	3410:
		stFolderCom.TaskBackGauge	:=eTask_BackGauge_AbsPos;
		stFolderCom.paraBackGauge	:=stFolder.BackGauge_M_ActPos+10;
		iSemiAutoStp	:=3411;
	3411:
		SA_Ton2(IN:=stFolderCom.TaskBackGauge = eTask_NULL , PT:=T#100MS , Q=> , ET=> );
		IF SA_Ton2.Q THEN
			SA_Ton2(IN:=FALSE);
			iSemiAutoStp	:=3420;
		END_IF	
	3420:
		stFolderCom.TaskClamp	:=eTask_ClampUnlock;
		stFolderCom.paraClamp	:=1;
		iSemiAutoStp	:=3421;
	3421:
		IF stFolderCom.TaskClamp = eTask_NULL THEN
			iSemiAutoStp	:=350;
		END_IF
		*)
(********************************************************************************)
	350:
		stFolderCom.TaskBackGauge	:=eTask_BackGauge_AbsPos;
		_ActBG_Target				:=SemiAuto_ActJob.BackGaugePos;
		stFolderCom.paraBackGaugeVelo	:= CNST_BACKGAUGE_SPEED_LOW;
		iSemiAutoStp	:=351;
	351:
		IF stFolderCom.TaskBackGauge = eTask_NULL THEN
			iSemiAutoStp	:=360;
		END_IF
	360:
		stFolderCom.TaskApron	:=eTask_ApronBtmFold_AbsPos;
		stFolderCom.ParaApronBtmFold	:=180;
		stFolderCom.paraApronFold_Auto	:=FALSE;
		iSemiAutoStp	:=361;
	361:
		IF stFolderCom.TaskApron = eTask_NULL THEN
			iSemiAutoStp	:=362;
		END_IF
	362:
		IF stFolder.Status.ApronBtmFold_AtHome THEN
			iSemiAutoStp	:=363;
		END_IF;
	363:
		stFolderCom.TaskClamp	:=eTask_ClampJog;
		IF _Contius OR (NOT _Contius AND rtPdlFold.Q) THEN
			iSemiAutoStp	:=370;
		END_IF
	370:
		//Out_GripperDatum_S0	:=Out_GripperDatum_S1	:=TRUE;		//insert to UNIT
		stFolderCom.TaskClamp	:=eTask_ClampLock;
		stFolderCom.paraClamp	:=6;
		iSemiAutoStp	:=371;
	371:
		IF stFolderCom.TaskClamp = eTask_NULL THEN
			iSemiAutoStp	:=372;
		END_IF
	372:
		IF SemiAuto_ActJob.ActType=1 THEN		//Close Squash
			iSemiAutoStp	:=380;
		ELSIF SemiAuto_ActJob.ActType=2 THEN	//Open Squash
			iSemiAutoStp	:=3800;
		END_IF
	380:
		ton372(IN:=TRUE , PT:=T#300MS , Q=> , ET=> );
		IF ton372.Q THEN
			iSemiAutoStp	:=500;
			ton372(IN:=FALSE);
		END_IF;
	//Open Squash Fun. 3800-3830
	3800:
		stFolderCom.TaskClamp	:=eTask_ClampUnlock;
		stFolderCom.paraClamp	:=1;
		iSemiAutoStp	:=3801;
	3801:
		IF stFolderCom.TaskClamp = eTask_NULL AND stFolder.ClampHt_ActPos>=stFolderPara.Clamp_MidPos  THEN
			iSemiAutoStp	:=3810;
		END_IF
	3810:
		stFolderCom.TaskBackGauge	:=eTask_BackGauge_AbsPos;
		IF SemiAuto_ActJob.FoldDir=0 THEN
			_tmp0	:=stFolderPara.SquashBackstop_OpenTop;
		ELSE
			_tmp0	:=stFolderPara.SquashBackstop_OpenBtm;
		END_IF
		_ActBG_Target				:=SemiAuto_ActJob.BackGaugePos-stFolderPara.SquashBackstop_External-_tmp0;
		stFolderCom.paraBackGaugeVelo	:= CNST_BACKGAUGE_SPEED_LOW;
		iSemiAutoStp	:=3811;
	3811:
		IF stFolderCom.TaskBackGauge = eTask_NULL THEN
			iSemiAutoStp	:=3820;
		END_IF
	3820:
		stFolderCom.TaskClamp	:=eTask_ClampLock;
		stFolderCom.paraClamp	:=6;
		iSemiAutoStp	:=3821;
	3821:
		IF stFolderCom.TaskClamp = eTask_NULL THEN
			iSemiAutoStp	:=380;
		END_IF


(*--------------------------------------------------------------------------*)
(*------------------------------分条功能开始--------------------------------*)	
(*--------------------------------------------------------------------------*)
	400:
	IF Hmi_bArray[62] THEN			//分条  + Slitter S.W.
		iSemiAutoStp	:=401;
	ELSE
		iSemiAutoStp	:=500;
	END_IF
	401:
		stFolderCom.TaskClamp	:=eTask_ClampJog;
		stFolder.SlitterRef		:=TRUE;
		IF stFolder.ClampHt_ActPos > stFolderPara.ClampHalfPos THEN
			stFolderCom.TaskBackGauge	:=eTask_BackGauge_AbsPos;
			_ActBG_Target				:=SemiAuto_ActJob.BackGaugePos;
			stFolderCom.paraBackGauge_GripType	:=SemiAuto_ActJob.GripType;
			stFolderCom.paraBackGaugeVelo	:= CNST_BACKGAUGE_SPEED_HIGH;
			bGripperDatumBack:=TRUE;
			iSemiAutoStp	:=402;
		END_IF
	402:
		IF stFolderCom.TaskBackGauge=eTask_NULL THEN
			iSemiAutoStp	:=410;
		END_IF
	410:
		Hmi_iArray[22]:=2 ;				//msg： Lock Grip
		IF stFolder.Status.Gripper THEN
			Hmi_iArray[22]:=0 ;
			iSemiAutoStp	:=420;
		END_IF;
	420:
		//Out_GripperDatum_S0	:=Out_GripperDatum_S1	:=TRUE;		//insert to UNIT
		stFolderCom.TaskClamp	:=eTask_ClampLock;
		stFolderCom.paraClamp	:=6;
		IF stFolder.Status.Clamp_AtPressPoint THEN
			iSemiAutoStp	:=430;
		END_IF
	430:
		stFolderCom.ParaApronBtmSlide := 0;
		stFolderCom.ParaApronTopSlide := 3;
		stFolderCom.TaskApron	:=eTask_ApronDaulSlide_AbsPos;
		iSemiAutoStp	:=431;
	431:
		IF stFolderCom.TaskApron = eTask_NULL THEN
			iSemiAutoStp	:=440;
		END_IF
	440:
		Hmi_iArray[22]:=7;				//msg： Operator Slitter
		stFolderCom.TaskSlitter	:=eTask_SlitterAct;
		iSemiAutoStp	:=441;
	441:
		IF stFolderCom.TaskSlitter	= eTask_NULL THEN
			iSemiAutoStp	:=450;
			Hmi_iArray[22]:=0;	
		END_IF
	450:
		stFolder.SlitterRef		:=FALSE;
		iSemiAutoStp	:=500;
(*--------------------------------------------------------------------------*)
(*----------------------------下一折弯角度 判断是否末JOB---------------------*)	
(*--------------------------------------------------------------------------*)
	500:
		IF SemiAuto_NextJob.FoldAngle <= 0 THEN
			iSemiAutoStp:=600;
//		ELSIF SemiAuto_NextJob.FoldAngle = 80 THEN 
//			iSemiAutoStp:=520;
		ELSE
			iSemiAutoStp:=510;
		END_IF;
	510:
//		IF SemiAuto_ActJob.GripType=SemiAuto_NextJob.GripType AND SemiAuto_ActJob.ReGrip=0 THEN 
		IF stFolderCom.paraBackGauge_GripType=SemiAuto_NextJob.GripType AND SemiAuto_ActJob.ReGrip=0 THEN	
			iSemiAutoStp	:=520;
		ELSE
			Hmi_iArray[22]:=1;				//msg： unLock Grip
			IF NOT stFolder.Status.Gripper THEN
				Hmi_iArray[22]	:=0;
				bGripperDatumBack:=FALSE;
				iSemiAutoStp	:=520;
			END_IF
		END_IF
	520:
		stFolderCom.TaskClamp	:=eTask_ClampUnlock;
		stFolderCom.paraClamp	:=SemiAuto_ActJob.UnClampHt;
		iSemiAutoStp	:=521;
	521:
		IF stFolderCom.TaskApron=eTask_NULL AND stFolderCom.TaskClamp = eTask_NULL THEN
			iSemiAutoStp	:=530;
		END_IF
	530:
		IF SemiAuto_ActJob.GripType=SemiAuto_NextJob.GripType THEN
			iSemiAutoStp	:=550;
		ELSE
			iSemiAutoStp	:=540;
		END_IF
	540:
		iSemiAutoStp	:=550;
		IF NOT stFolder.Status.Gripper THEN
			stFolderCom.TaskBackGauge	:=eTask_BackGauge_BackPos;
			_ActBG_Target				:=SemiAuto_NextJob.BackGaugePos;
			stFolderCom.paraBackGauge_GripType	:=SemiAuto_NextJob.GripType;
			stFolderCom.paraBackGaugeVelo	:= CNST_BACKGAUGE_SPEED_HIGH;
			stFolderCom.paraBackGauge_GripOPEN	:=FALSE;
			bGripperDatumBack:=FALSE;
			iSemiAutoStp	:=541;
		END_IF
	541:
		IF stFolderCom.TaskBackGauge = eTask_NULL AND ton541.Q THEN
			iSemiAutoStp	:=550;
		END_IF
		
		
	550:	//本折弯结束,跳转到下一JOB
		
		iSemiAuto_JobId:=iSemiAuto_JobId+1;
		IF SemiAuto_ActJob.ActType=0 THEN
			Hmi_iArray[70]	:=Hmi_iArray[70]+1;
		END_IF
		iSemiAutoStp	:=50;
(*--------------------------------------------------------------------------*)
(*--------------------------------------所有JOB工作完成---------------------*)	
(*--------------------------------------------------------------------------*)
	600:	//所有JOBID完成,结束
		Hmi_iArray[22]:=1;			//msg:	Unlock Gripper
		TONDELAY(IN:= TRUE , PT:=GRIP_AUTOOPEN_TIME , Q=> , ET=> );
		IF stFolderPara.swClampOpen_InAuto AND TONDELAY.Q THEN
			stFolderCom.paraBackGauge_Grip :=1;
			Hmi_iArray[22]	:=0;
		END_IF
		IF NOT stFolder.Status.Gripper THEN
			Hmi_iArray[22]:=0;
			stFolderCom.TaskClamp	:=eTask_ClampUnlock;
			stFolderCom.paraClamp	:=2;
			iSemiCount:=iSemiCount+1;
			Hmi_iArray[70]	:=Hmi_iArray[70]+1;
			iSemiAutoStp	:=601;
			TONDELAY(IN := FALSE);  // 复位定时器输入，准备下次启动
		END_IF
	601:
		IF stFolderCom.TaskClamp = eTask_NULL THEN
			IF stFolderPara.swFeedMechanism THEN
				iSemiAutoStp	:=700;
			ELSE
				iSemiAutoStp	:=1;
			END_IF
			iSemiAuto_JobId	:=0;
		END_IF
(*--------------------------------------------------------------------------*)
(*--------------------------------------开始进料工作------------------------*)	
(*--------------------------------------------------------------------------*)		
	700:
		FeedEnable:=TRUE;
		A_FeedAuto();
		tonFeed(IN:=FeedDone , PT:=T#1S , Q=> , ET=> );
		IF tonFeed.Q THEN
			FeedEnable:=FALSE;
			iFeedAutoStep:=0;
			iSemiAutoStp:=4;	
		END_IF
(*--------------------------------------------------------------------------*)
(*--------------------------------------翻转--------------------------------*)
(*--------------------------------------------------------------------------*)		
	800:
		IF SemiAuto_ActJob.ActType=8 THEN			//翻转开关
			stFolder.Status.Flip_AtWork := TRUE;
			iSemiAutoStp	:=810;
		ELSE
			iSemiAutoStp	:=500;
		END_IF
	801:
		stFolderCom.TaskClamp	:=eTask_ClampUnlock;
		stFolderCom.paraClamp	:=4;
		IF stFolder.ClampHt_ActPos > stFolderPara.ClampHalfPos THEN
			stFolderCom.TaskBackGauge	:=eTask_BackGauge_AbsPos;
			_ActBG_Target				:=SemiAuto_ActJob.BackGaugePos+50;
			stFolderCom.paraBackGaugeVelo	:= CNST_BACKGAUGE_SPEED_HIGH;
//			bGripperDatumBack:=TRUE;
			iSemiAutoStp	:=802;
		END_IF
	802:
		IF stFolderCom.TaskBackGauge = eTask_NULL AND stFolder.BackGauge_T2_ActPos >= _ActBG_Target THEN
			iSemiAutoStp	:=810;
		END_IF
	810:
		stFolderCom.paraBackGauge_Grip := 1;
		IF NOT stFolder.Status.Gripper THEN
		
			iSemiAutoStp	:=811;
		END_IF
		
	811:
		stFolderCom.TaskClamp	:=eTask_ClampUnlock;
		stFolder.Status.Clamp_Slow := TRUE;
		stFolderCom.paraClamp	:=70;
		IF stFolder.ClampHt_ActPos > 70 THEN
			stFolderCom.TaskClamp :=eTask_NULL;
			stFolder.Status.Clamp_Slow := FALSE;
			iSemiAutoStp	:=812;
		END_IF
	812:
		ton812(IN:= iSemiAutoStp =812, PT:=T#1000MS , Q=> , ET=> );
		IF ton812.Q THEN
			stFolderCom.ParaApronBtmSlide := 2;
			stFolderCom.ParaApronTopSlide := 0;
			stFolderCom.TaskApron	:=eTask_ApronDaulSlide_AbsPos;
			iSemiAutoStp	:=813;
		END_IF
	813:
		IF stFolderCom.TaskApron = eTask_NULL THEN
//			stFolderCom.TaskTable	:=	eTask_NULL;
			Ton813(IN:=stFolderCom.TaskApron =	eTask_NULL, PT:=T#1000MS , Q=> , ET=> );
			IF ton813.Q THEN
//				stFolderCom.TaskTable		:=eTask_Table_AbsPos;
//	 			stFolderCom.paraTablePos	:=480;				//吸板位置
				iSemiAutoStp	:=820;
				Ton813(IN:=FALSE );
			END_IF
		END_IF
		
	814:
		stFolderCom.TaskTable	:=	eTask_NULL;
		ton814(IN:=iSemiAutoStp =814 , PT:=T#500MS , Q=> , ET=> );
		IF ton814.Q THEN
			iSemiAutoStp	:=820;
		END_IF
	820:
		stFolderCom.TaskTable		:=eTask_Table_AbsPos;
	 	stFolderCom.paraTablePos	:=470;				//吸板位置
		IF stFolder.Table_ActPos > 100 THEN
			iSemiAutoStp	:=821;
		END_IF
		Tonagain(IN:=stFolderCom.TaskTable = eTask_Table_AbsPos AND stFolder.Table_ActPos < 10, PT:=T#500MS , Q=> , ET=> );
		IF Tonagain.Q THEN
			iSemiAutoStp	:=814;
		END_IF
		
	821:
		IF stFolder.Table_ActPos >= 450 AND SemiAuto_ActJob.FoldDir=1 THEN
			stFolderCom.TaskApron			:=eTask_ApronTopFold_AbsPos;
			stFolderCom.ParaApronTopFold	:=73;
			stFolderCom.paraApronFold_Auto	:=TRUE;
			stFolder.Status.Flip_WorkDone 	:=TRUE;
			stFolderCom.TaskTable			:=	eTask_NULL;
			stFolderCom.TaskBackGauge	:=eTask_BackGauge_AbsPos;
			_ActBG_Target				:=SemiAuto_ActJob.BackGaugePos+300;
			stFolderCom.paraBackGaugeVelo	:= CNST_BACKGAUGE_SPEED_HIGH;
			bGripperDatumBack:=FALSE;
			stFolderCom.paraBackGauge_GripType	:=SemiAuto_NextJob.GripType;
			iSemiAutoStp	:=822;
		END_IF;
		
	822:
		IF stFolder.ApronTop_Fold_ActAngle > 105 AND NOT FeedDemoMode THEN
			stFolderCom.paraFlip_SuctionCup := 1;
		END_IF;
		ton822(IN:= stFolderCom.paraFlip_SuctionCup = 1 OR FeedDemoMode, PT:=T#800MS , Q=> , ET=> );
		IF TON822.Q THEN
			stFolder.Status.Flip_WorkDone 	:=FALSE;
			Ton822(IN:=FALSE );
			IF FeedDemoMode THEN
				iSemiAutoStp	:=825;
			ELSE
				iSemiAutoStp	:=823;
			END_IF
//			iSemiAutoStp	:=823;
		END_IF
	823:
		Ton823(IN:=stFolderCom.TaskApron = eTask_NULL , PT:=T#500MS , Q=> , ET=> );
		IF stFolderCom.TaskApron = eTask_NULL AND TON823.Q
			AND ((semiAuto_ActJob.FoldDir = 0 AND In_sigBtmApron_SlideFWD) OR (semiAuto_ActJob.FoldDir = 1 AND In_sigTopApron_SlideFWD)) THEN
			Ton823(IN:=FALSE );
			stFolderCom.TaskClamp	:=eTask_ClampLock;
			stFolderCom.paraClamp	:=50;
//			stFolderCom.paraFlip_SuctionCup := 0;
			iSemiAutoStp	:=824;
		END_IF
	824:
		IF stFolder.ClampHt_ActPos < 60 THEN
			stFolderCom.TaskClamp		:=eTask_NULL;
			stFolderCom.paraFlip_SuctionCup := 0;
		END_IF
		IF NOT stFolder.Status.FlipSuctionCup THEN
			stFolderCom.TaskTable		:=eTask_Table_AbsPos;
	 		stFolderCom.paraTablePos	:=750;
			iSemiAutoStp	:=825;
		END_IF
	825:
		Ton825(IN:=iSemiAutoStp =825 , PT:=T#2000MS , Q=> , ET=> );
		IF stFolderCom.TaskTable = eTask_NULL AND ton825.q THEN
			stFolderCom.TaskTable		:=eTask_Table_AbsPos;
	 		stFolderCom.paraTablePos	:=0;
			Ton825(IN:=FALSE );
			iSemiAutoStp	:=830;
		END_IF	
	830:
		IF stFolderCom.TaskTable = eTask_NULL AND stFolder.Status.Table_AtHome THEN
			stFolderCom.TaskTable			:=	eTask_NULL;
//			bGripperDatumBack:=FALSE;

			stFolderCom.TaskBackGauge	:=eTask_BackGauge_AbsPos;
			_ActBG_Target				:=SemiAuto_NextJob.BackGaugePos-50;
			stFolderCom.paraBackGaugeVelo	:= CNST_BACKGAUGE_SPEED_HIGH;
			iSemiAutoStp	:=831;
		END_IF
	831:
		IF stFolderCom.TaskBackGauge=eTask_NULL THEN
			stFolderCom.paraBackGauge_Grip := 0;
//			bGripperDatumBack:=TRUE;
			iSemiAutoStp	:=832;
		END_IF
	832:	
		IF stFolder.Status.Gripper THEN
			stFolder.Status.Flip_AtWork := FALSE;
			iSemiAutoStp	:=500;
		END_IF
END_CASE
END_ACTION

ACTION A_SlitterAuto:

IF rtSlitterMode.Q THEN 
	i114:=i114+1;
END_IF

IF rtSlitterMode.Q THEN
	iSlitterAutoStp			:=0;
	SlitterAuto_iJobId		:=0;
	SlitterAuto_iPieceNum	:=0;
	stFolder.SlitterRef		:=TRUE;
	_ActBG_Target	:=0;
	SlitterAuto_rWidthOdd	:=0;
	
	
	stFolderCom.TaskClamp		:=eTask_NULL;
	stFolderCom.TaskBackGauge	:=eTask_NULL;
	stFolderCom.TaskApron		:=eTask_NULL;
	stFolderCom.TaskSlitter		:=eTask_NULL;
	stFolderCom.TaskTable		:=eTask_NULL;
END_IF

(*******************************************************************************)
(***************************** Start Slitter Auto Job *****************************)
(*******************************************************************************)
SlitterAuto_ActJob_Width	:=Hmi_rSlitter[SlitterAuto_iJobId+10];
SlitterAuto_ActJob_Num		:=Hmi_rSlitter[SlitterAuto_iJobId+22];

Hmi_iArray[80]	:=TO_UINT(SlitterAuto_iPieceNum);
tmp2:=TO_INT(Hmi_rSlitter[2]-1);
Hmi_iArray[81]	:=REAL_TO_UINT(Hmi_rSlitter[LIMIT(0,SlitterAuto_iJobId,tmp2)+22]);
Hmi_iArray[82]	:= TO_UINT(SlitterAuto_iJobId);

IF rtSlitterMode.Q THEN
	stFolderCom.TaskBackGauge	:=eTask_NULL;
	iSlitterAutoStp	:=0;
END_IF

CASE iSlitterAutoStp OF
	0:
		stFolderCom.TaskClamp	:=eTask_ClampJog;
		IF rtSlitterMode.Q AND Hmi_rSlitter[2]>0 THEN		(*Slitter Auto Start*)
			iSlitterAutoStp	:=1;
		END_IF
	1:
		bSlitterHead	:=Hmi_bArray[81] AND Hmi_rSlitter[1]>0;		//边料在前,且有边角料
		Out_Gripper	:=Out_Gripper2	:=FALSE;
		IF NOT stFolder.Status.Gripper AND NOT stFolder.Status.Gripper2 THEN
			iSlitterAutoStp	:=2;
		END_IF
	2:
		stFolderCom.TaskClamp	:=eTask_ClampUnlock;
		stFolderCom.paraClamp	:=2;
		iSlitterAutoStp	:=3;
	3:
		IF NOT stFolder.Status.BG_Coupled
			AND NOT stFolder.Status.Clamp_LtHalfPoint THEN
			stFolderCom.TaskBackGauge	:=eTask_BackGauge_GearIn;
			iSlitterAutoStp	:=4;
		ELSE
			iSlitterAutoStp	:=5;
		END_IF;
	4:
		IF stFolderCom.TaskBackGauge=eTask_NULL THEN
			iSlitterAutoStp	:=5;
		END_IF
	5:
		IF NOT stFolder.Status.Clamp_LtHalfPoint THEN
			stFolderCom.TaskBackGauge	:=eTask_BackGauge_AbsPos;
			stFolderCom.paraBG_T1	:=stFolderPara.BackGaugeMaxPos;
			stFolderCom.paraBackGauge_GripType	:=2;
			stFolderCom.paraBackGaugeVelo	:=CNST_BACKGAUGE_SPEED_HIGH;
			iSlitterAutoStp	:=6;
		END_IF
	6:
		iSlitterAutoStp	:=7;
	7:
		IF stFolderCom.TaskClamp = eTask_NULL AND stFolderCom.TaskBackGauge=eTask_NULL THEN
			iSlitterAutoStp	:=10;
		END_IF
	10:	
		stFolderCom.TaskClamp	:=eTask_ClampJog;
		IF bSlitterHead THEN		//Odd. Before or After.
			SlitterAuto_rWidthOdd	:=Hmi_rSlitter[0] - Hmi_rSlitter[1];
		ELSE
			SlitterAuto_rWidthOdd	:=Hmi_rSlitter[0] - SlitterAuto_ActJob_Width;
		END_IF
		_ActBG_Target	:=SlitterAuto_rWidthOdd;
		IF  stFolder.ClampHt_ActPos > stFolderPara.Clamp_LowPos THEN
			stFolderCom.TaskBackGauge	:=eTask_BackGauge_AbsPos;
			stFolderCom.paraBG_T1	:=_ActBG_Target;
			stFolderCom.paraBackGauge_GripType	:=2;
			iSlitterAutoStp	:=11;
		END_IF
	11:
		IF stFolderCom.TaskBackGauge=eTask_NULL THEN
			iSlitterAutoStp	:=20;
		END_IF
	20:
		stFolderCom.ParaApronBtmSlide := 0;
		stFolderCom.ParaApronTopSlide := 3;
		stFolderCom.TaskApron	:=eTask_ApronDaulSlide_AbsPos;
		iSlitterAutoStp	:=21;
	21:
		IF stFolderCom.TaskApron = eTask_NULL THEN
			iSlitterAutoStp	:=30;
		END_IF
	30:	(*放入板材,夹住板材,压紧板材*)
		stFolderCom.TaskClamp	:=eTask_ClampJog;
		IF (NOT stFolder.Status.Clamp_LtHalfPoint) THEN
			IF Hmi_bArray[82] THEN				//Load Material S.W.
				iSlitterAutoStp	:=32;
			END_IF;
		END_IF;
		IF stFolder.Status.Gripper  THEN
			iSlitterAutoStp	:=100;
		END_IF
(*************************** Load Material Function *******************************)
	32:
		stFolderCom.TaskApron			:=eTask_ApronBtmFold_AbsPos;
		stFolderCom.ParaApronBtmFold	:=90;
		stFolderCom.paraApronFold_Auto	:=FALSE;
		iSlitterAutoStp	:=33;
	33:
		IF stFolderCom.TaskApron = eTask_NULL THEN
			iSlitterAutoStp	:=34;
		END_IF
	34:
		stFolderCom.TaskClamp	:=eTask_ClampJog;
		IF stFolder.Status.Gripper THEN
			iSlitterAutoStp	:=50;
		END_IF;
		IF Hmi_bArray[82] THEN					//Load Material S.W.
			stFolderCom.TaskApron			:=eTask_ApronBtmFold_AbsPos;
			stFolderCom.ParaApronBtmFold	:=180;
			stFolderCom.paraApronFold_Auto	:=FALSE;
			iSlitterAutoStp	:=35;
		END_IF;
	35:
		IF stFolderCom.TaskApron = eTask_NULL THEN
			iSlitterAutoStp	:=40;
		END_IF;
(*********************************************************************************)
	40:
		stFolderCom.TaskClamp	:=eTask_ClampJog;
		Hmi_iArray[22]:=Hmi_iArray[22] OR 16#0002; ;	//Operation message
		IF stFolder.Status.Gripper THEN
			Hmi_iArray[22]:=Hmi_iArray[22] AND 16#FFFD;	//Operation message
			iSlitterAutoStp	:=100;
		END_IF;
(*********************** Put Down ApronBtmFold**********************************)
	50:
		stFolderCom.TaskApron			:=eTask_ApronBtmFold_AbsPos;
		stFolderCom.ParaApronBtmFold	:=180;
		stFolderCom.paraApronFold_Auto	:=FALSE;
		iSlitterAutoStp	:=51;
	51:
		IF stFolderCom.TaskApron = eTask_NULL THEN
			iSlitterAutoStp	:=100;
		END_IF;
(**************************** Start Loop *************************************)
	100:
		stFolderCom.TaskClamp	:=eTask_ClampLock;
		stFolderCom.paraClamp	:=6;
		iSlitterAutoStp	:=101;
	101:
		IF stFolderCom.TaskClamp = eTask_NULL THEN
			iSlitterAutoStp	:=110;
			stFolderCom.TaskApron	:=0;
		END_IF
	110:
		stFolderCom.TaskSlitter	:=eTask_SlitterAct;
		Hmi_iArray[22]:=7;			//msg： Operator Slitter
		iSlitterAutoStp	:=120;
	120:
		stFolderCom.TaskClamp	:=eTask_ClampJog;
		IF stFolderCom.TaskSlitter	= eTask_NULL THEN
			Hmi_iArray[22]:=0;
			IF NOT bSlitterHead THEN
				SlitterAuto_iPieceNum	:=SlitterAuto_iPieceNum+1;
			END_IF
			bSlitterHead	:=FALSE;
			iSlitterAutoStp	:=130;
		END_IF
(*
	130:
		IF (SlitterAuto_iPieceNum >= SlitterAuto_ActJob_Num)  
			OR ( (Hmi_bArray[81] OR SlitterAuto_rWidthOdd<=SlitterAuto_ActJob_Width )
				 AND (SlitterAuto_iJobId+1) >= Hmi_rSlitter[2] AND (SlitterAuto_iPieceNum+1) >= SlitterAuto_ActJob_Num) THEN
			SlitterAuto_iJobId	:=SlitterAuto_iJobId+1;
			SlitterAuto_iPieceNum	:=0;
		END_IF
		IF (Hmi_bArray[81] AND (SlitterAuto_iJobId+1) >= Hmi_rSlitter[2] AND 1= SlitterAuto_ActJob_Num) THEN
			SlitterAuto_iJobId	:=SlitterAuto_iJobId+1;
		
		END_IF
		iSlitterAutoStp	:=131;
*)
	130:
		IF (SlitterAuto_iPieceNum >= SlitterAuto_ActJob_Num) THEN
			SlitterAuto_iJobId	:=SlitterAuto_iJobId+1;
			SlitterAuto_iPieceNum	:=0;
		ELSIF ( Hmi_bArray[81] AND (SlitterAuto_iJobId+1) >= Hmi_rSlitter[2] AND (SlitterAuto_iPieceNum+1) >= SlitterAuto_ActJob_Num)
			OR ((Hmi_rSlitter[1]=0 ) AND (SlitterAuto_iJobId+1) >= Hmi_rSlitter[2] AND (SlitterAuto_iPieceNum+1) >= SlitterAuto_ActJob_Num) THEN
			SlitterAuto_iJobId	:=SlitterAuto_iJobId+1;
		END_IF
		iSlitterAutoStp	:=131;
	131:
		iSlitterAutoStp	:=132;
	132:
		iSlitterAutoStp	:=140;
		(*
	140:
		IF (SlitterAuto_iJobId >= Hmi_rSlitter[2]) OR 
				(Hmi_bArray[81] AND SlitterAuto_iJobId+1 >= Hmi_rSlitter[2] AND (SlitterAuto_iPieceNum+1) >= SlitterAuto_ActJob_Num) THEN 
			iSlitterAutoStp	:=200;
		ELSE
			iSlitterAutoStp	:=150;
		END_IF		*)
	140:
		IF (SlitterAuto_iJobId >= Hmi_rSlitter[2])
			OR (Hmi_bArray[81] AND (SlitterAuto_iJobId+1) >= Hmi_rSlitter[2] AND (SlitterAuto_iPieceNum+1) >= SlitterAuto_ActJob_Num)
			OR ((Hmi_rSlitter[1]=0 ) AND (SlitterAuto_iJobId+1) >= Hmi_rSlitter[2] AND (SlitterAuto_iPieceNum+1) >= SlitterAuto_ActJob_Num)
 		THEN 
			iSlitterAutoStp	:=200;
		ELSE
			iSlitterAutoStp	:=150;
		END_IF	
	150:
		stFolderCom.TaskClamp	:=eTask_ClampUnlock;
		stFolderCom.paraClamp	:=0;
		iSlitterAutoStp	:=151;
	151:
		IF stFolderCom.TaskClamp = eTask_NULL THEN
			iSlitterAutoStp	:=160;
		END_IF
	160:
		SlitterAuto_rWidthOdd	:= SlitterAuto_rWidthOdd - SlitterAuto_ActJob_Width;
		_ActBG_Target	:= SlitterAuto_rWidthOdd; 
		stFolderCom.TaskBackGauge	:=eTask_BackGauge_AbsPos;
		stFolderCom.paraBG_T1	:=_ActBG_Target;
		stFolderCom.paraBackGauge_GripType	:=2;
		stFolderCom.paraBackGaugeVelo	:=CNST_BACKGAUGE_SPEED_HIGH;
		iSlitterAutoStp	:=161; 
	161:
		IF stFolderCom.TaskBackGauge=eTask_NULL THEN
			iSlitterAutoStp	:=100;
		END_IF

(**************************** Finish Work *************************************)		
	200:
		Hmi_iArray[22]:=1;			//msg:	Unlock Gripper
		IF NOT stFolder.Status.Gripper THEN
			Hmi_iArray[22]:=0;
			stFolderCom.TaskClamp	:=eTask_ClampUnlock;
			stFolderCom.paraClamp	:=2;
			iSlitterAutoStp	:=201;
		END_IF
	201:
		IF stFolderCom.TaskClamp = eTask_NULL THEN
			iSlitterAutoStp	:=1;
			SlitterAuto_iJobId	:=0;
			SlitterAuto_iPieceNum	:=0;
		END_IF
		
		
	
END_CASE
END_ACTION

ACTION aWarning:
IF NOT In_EMG_RopeStop THEN
	Hmi_iArray[26]:=Hmi_iArray[26] OR 16#0001; ;	//Rope Limit
ELSIF In_EMG_RopeStop THEN
	Hmi_iArray[26]:=Hmi_iArray[26] AND 16#FFFE; ;	//Rope Limit
END_IF

IF In_sigPumpJam THEN
	Hmi_iArray[26]:=Hmi_iArray[26] OR 16#0002; ;	//PumpJamAlarm
ELSIF NOT In_sigPumpJam THEN
	Hmi_iArray[26]:=Hmi_iArray[26] AND 16#FFFD; ;	//PumpJamAlarm
END_IF

IF In_sigLubeJam THEN
	Hmi_iArray[26]:=Hmi_iArray[26] OR 16#0004; ;	//LubeJamAlarm
ELSIF NOT In_sigLubeJam THEN
	Hmi_iArray[26]:=Hmi_iArray[26] AND 16#FFFB; ;	//LubeJamAlarm
END_IF;

IF In_EMG_MainCabinet THEN
	Hmi_iArray[26]:=Hmi_iArray[26] OR 16#0008; ;	//Electric Cabinet EMG
ELSIF NOT In_EMG_MainCabinet THEN
	Hmi_iArray[26]:=Hmi_iArray[26] AND 16#FFF7; ;	//Electric Cabinet EMG
END_IF;

IF In_EMG_HandleCabinet THEN
	Hmi_iArray[26]:=Hmi_iArray[26] OR 16#0010; ;	//Handling Cabinet EMG
ELSIF NOT In_EMG_HandleCabinet THEN
	Hmi_iArray[26]:=Hmi_iArray[26] AND 16#FFEF; ;	//Handling Cabinet EMG
END_IF;
END_ACTION

ACTION DualPump:
(********* Relation Map   Freq and Num******************************************************
5HZ-----71		6HZ----86		7.5HZ---107
10HZ--143		20HZ--286		30HZ--428
40HZ---571		50HZ--714		60HZ--857
70HZ---1000
*******************************************************************)

rPropCmd_BtmSlide	:=0;
rPropCmd_BtmFold	:=0;
rPropCmd_ClampUp	:=0;
rPropCmd_ClampDown	:=0;
rPropCmd_TopSlide	:=0;
rPropCmd_TopFold	:=0;

IF Out_ApronTop_SlideFWD THEN
	stFolder.PumpA_SetVal	:=SEL(stFolder.Status.ApronTopSlide_AtSlow, CNST_APRON_TOPSLIDE_FWD_SPD,CNST_APRON_TOPSLIDE_FWD_CREEP_SPD);		//540
	rPropCmd_TopSlide	:=-CNST_APRON_TOPSLIDE_FWD_SPD;
	//stFolder.PumpB_SetVal	:=143;
ELSIF Out_ApronTop_SlideBWD THEN
	stFolder.PumpA_SetVal	:=SEL(stFolder.Status.ApronTopSlide_AtSlow, CNST_APRON_TOPSLIDE_BWD_SPD,CNST_APRON_TOPSLIDE_BWD_CREEP_SPD);		//428
	rPropCmd_TopSlide	:=CNST_APRON_TOPSLIDE_BWD_SPD;
	//stFolder.PumpB_SetVal	:=143;
END_IF;

IF Out_ApronBtm_SlideFWD THEN
	//stFolder.PumpA_SetVal	:=143;
//	tmp1	:=SEL(Out_SlitterFwd OR Out_SlitterBwd,CNST_APRON_BTMSLIDE_FWD_SPD,CNST_APRON_BTMSLIDE_FWD_CREEP_SPD);
	stFolder.PumpB_SetVal	:=SEL(stFolder.Status.ApronBtmSlide_AtSlow OR GVL.gvl_bSlipPatch_BtmSlide, CNST_APRON_BTMSLIDE_FWD_SPD,CNST_APRON_BTMSLIDE_FWD_CREEP_SPD);
	rPropCmd_BtmSlide	:=-CNST_APRON_BTMSLIDE_FWD_SPD;
ELSIF Out_ApronBtm_SlideBWD THEN
	//stFolder.PumpA_SetVal	:=143;
	stFolder.PumpB_SetVal	:=SEL(stFolder.Status.ApronBtmSlide_AtSlow, CNST_APRON_BTMSLIDE_BWD_SPD,CNST_APRON_BTMSLIDE_BWD_CREEP_SPD);	//428
	rPropCmd_BtmSlide	:=CNST_APRON_BTMSLIDE_BWD_SPD;
END_IF;
IF Out_ApronTop_FoldFWD THEN
	stFolder.PumpB_SetVal	:=CNST_HYD_IDLE_SPD;
	stFolder.PumpA_SetVal	:=SEL(stFolder.Status.ApronFold_AtSlow, CNST_APRON_TOPFOLD_FWD_SPD,CNST_APRON_TOPFOLD_FWD_CREEP_SPD);
	rPropCmd_TopFold	:=-CNST_APRON_TOPFOLD_FWD_SPD;
ELSIF Out_ApronTop_FoldBWD THEN
	stFolder.PumpB_SetVal	:=CNST_HYD_IDLE_SPD;
	stFolder.PumpA_SetVal	:=SEL(stFolder.Status.ApronFold_AtSlow, CNST_APRON_TOPFOLD_BWD_SPD,CNST_APRON_TOPFOLD_BWD_CREEP_SPD);
	rPropCmd_TopFold	:=CNST_APRON_TOPFOLD_BWD_SPD;
ELSIF Out_ApronBtm_FoldFWD THEN
	stFolder.PumpB_SetVal	:=SEL(stFolder.Status.ApronFold_AtSlow, CNST_APRON_BTMFOLD_FWD_SPD,CNST_APRON_BTMFOLD_FWD_CREEP_SPD);
	stFolder.PumpA_SetVal	:=CNST_HYD_IDLE_SPD;
	rPropCmd_BtmFold	:=CNST_APRON_BTMFOLD_FWD_SPD;
ELSIF Out_ApronBtm_FoldBWD THEN
	stFolder.PumpB_SetVal	:=SEL(stFolder.Status.ApronFold_AtSlow OR gvl_bSlipPatch_BtmFold, CNST_APRON_BTMFOLD_BWD_SPD,CNST_APRON_BTMFOLD_BWD_CREEP_SPD);
	stFolder.PumpA_SetVal	:=CNST_HYD_IDLE_SPD;
	rPropCmd_BtmFold	:=-CNST_APRON_BTMFOLD_BWD_SPD;
ELSIF Out_ClampUp AND (stFolder.Status.Clamp_LtHalfPoint OR stFolder.Status.Clamp_Slow) AND (fbUnitModeManager.eModeStatus<>ePMLProtUnitMode_Manual) THEN
	stFolder.PumpA_SetVal	:=CNST_HYD_IDLE_SPD;
	stFolder.PumpB_SetVal	:=CNST_HYD_IDLE_SPD;
	rPropCmd_ClampUp	:=CNST_CLAMP_OPEN_SPD_LT_HALF;
ELSIF Out_ClampUp AND stFolder.Status.Clamp_LtHalfPoint AND (fbUnitModeManager.eModeStatus=ePMLProtUnitMode_Manual) THEN
	stFolder.PumpA_SetVal	:=CNST_CLAMP_OPEN_SPD_LT_HALF;
	stFolder.PumpB_SetVal	:=CNST_CLAMP_OPEN_SPD_LT_HALF;
	rPropCmd_ClampUp	:=CNST_CLAMP_OPEN_SPD_LT_HALF;
ELSIF Out_ClampUp AND (NOT stFolder.Status.Clamp_LtHalfPoint ) THEN
	stFolder.PumpA_SetVal	:=CNST_CLAMP_OPEN_SPD_GT_HALF;
	stFolder.PumpB_SetVal	:=CNST_CLAMP_OPEN_SPD_GT_HALF;
	rPropCmd_ClampUp	:=CNST_CLAMP_OPEN_SPD_GT_HALF;
//ELSIF Out_ClampDown AND stFolder.Status.Clamp_AtPressPoint THEN
//	stFolder.PumpA_SetVal	:=119;
//	stFolder.PumpB_SetVal	:=119;
ELSIF Out_ClampDown AND (stFolder.Status.Clamp_LtHalfPoint OR stFolder.Status.Clamp_Slow) THEN
	stFolder.PumpA_SetVal	:=CNST_CLAMP_CLOSE_SPD_LT_HALF;
	stFolder.PumpB_SetVal	:=CNST_CLAMP_CLOSE_SPD_LT_HALF;
	rPropCmd_ClampDown	:=CNST_CLAMP_CLOSE_SPD_LT_HALF;
	//stFolder.PumpA_SetVal	:=143;
	//stFolder.PumpB_SetVal	:=143;
ELSIF Out_ClampDown AND (NOT stFolder.Status.Clamp_LtHalfPoint) THEN
	stFolder.PumpA_SetVal	:=CNST_CLAMP_CLOSE_SPD_GT_HALF;
	stFolder.PumpB_SetVal	:=CNST_CLAMP_CLOSE_SPD_GT_HALF;
	rPropCmd_ClampDown	:=CNST_CLAMP_CLOSE_SPD_GT_HALF;
ELSIF Out_GaugingF_Ext OR Out_GaugingF_Rtn	OR Out_GaugingR_Ext	OR Out_GaugingR_Rtn THEN
	stFolder.PumpB_SetVal	:=428;
END_IF



(*
Short Vertical Light Curtain is ON,  =>  Slitter Slow down.
Long Vertical Light Curtain is ON,  =>  All Action Slow down.
Horizontal Light Curtain is ON,  =>  Apron Slide or Fold Stop,Slitter Slow down.
Long Vertical and Horizontal Light Curtain is ON,  =>  Apron Folder Slow down..
Long Vertical Light Curtain and Laser is ON,  =>  All Action Stop.  cancel Laser Action Continue.
*)

//IF (Out_ApronTop_SlideFWD OR Out_ApronTop_SlideBWD OR (Out_ApronBtm_SlideFWD AND NOT Out_SlitterFwd AND NOT Out_SlitterBwd) OR Out_ApronBtm_SlideBWD ) AND (NOT In_sigLC_H) THEN
//	_override	:=0;
//ELSIF ( Out_SlitterFwd OR Out_SlitterBwd ) AND ( NOT In_sigLC_VShort OR NOT In_sigLC_VLong ) THEN
//	_override	:=20;
//ELSIF (Out_ApronTop_FoldFWD OR Out_ApronTop_FoldBWD OR Out_ApronBtm_FoldFWD OR Out_ApronBtm_FoldBWD) AND (NOT In_sigLC_VLong AND NOT In_sigLC_H) THEN
//	_override	:=20;
//ELSIF (Out_ApronTop_SlideFWD OR Out_ApronTop_SlideBWD OR Out_ApronBtm_SlideFWD OR Out_ApronBtm_SlideBWD ) AND (NOT In_sigLC_VLong) THEN
//	_override	:=20;
//ELSIF Out_ClampDown AND ( NOT In_sigLC_VShort OR NOT In_sigLC_VLong OR NOT In_sigLC_H) THEN
//	_override	:=20;
//ELSE
//	_override	:=100;
//END_IF
b_sigLC_VShort	:=NOT In_sigLC_VShort;
IF NOT In_swLC_Enable THEN
	_override	:=100;
	b_sigLC_VShort	:=FALSE;
END_IF;
//Enable SW can't Close Laser.
IF Out_ClampDown AND (NOT Hmi_bArray[12] AND In_sigLaserFinger AND NOT In_sigClampMute) THEN
	_override	:=0;
END_IF;
(*************************************************************************************************************)
//IF gblTon THEN
//	stFolder.PumpA_SetVal	:=118;
//	stFolder.PumpB_SetVal	:=118;
//END_IF

IF _override=0 THEN
	_PumpA_SetVal	:=0;
	_PumpB_SetVal	:=0;
ELSIF stFolder.PumpA_SetVal<10 AND stFolder.PumpB_SetVal<10 THEN
	_PumpA_SetVal	:=stFolder.PumpA_SetVal;
	_PumpB_SetVal	:=stFolder.PumpB_SetVal;
ELSE 
	_PumpA_SetVal	:=LIMIT(100,stFolder.PumpA_SetVal * _override /100,1000);
	_PumpB_SetVal	:=LIMIT(100,stFolder.PumpB_SetVal * _override /100,1000);
END_IF


Ton_DP0(IN:=(NOT Out_ClampDown AND NOT Out_ClampUp 
			AND NOT Out_ApronTop_SlideFWD AND NOT Out_ApronTop_SlideBWD AND NOT Out_ApronBtm_FoldFWD AND NOT Out_ApronBtm_FoldBWD
			AND stFolder.PumpA_SetVal<>PUMP_FREQ_IDLE) , PT:=T#5S);
Ton_DP1(IN:=(NOT Out_ClampDown AND NOT Out_ClampUp
			AND NOT Out_ApronTop_FoldFWD AND NOT Out_ApronTop_FoldBWD AND NOT Out_ApronBtm_SlideFWD AND NOT Out_ApronBtm_SlideBWD
			AND NOT Out_GaugingF_Ext AND NOT Out_GaugingF_Rtn AND NOT Out_GaugingR_Ext AND NOT Out_GaugingR_Rtn
			AND stFolder.PumpB_SetVal<>PUMP_FREQ_IDLE) , PT:=T#5S);	
IF Ton_DP0.Q THEN
	_PumpA_SetVal	:=PUMP_FREQ_IDLE;
END_IF
IF Ton_DP1.Q THEN
	_PumpB_SetVal	:=PUMP_FREQ_IDLE;
END_IF


(**********************************  RopeStop Emgerence ,  *************************************)
tonRopeStop(IN:= NOT In_EMG_RopeStop AND stFolder.Status.ApronBtmFold_AtHome , PT:=T#3S , Q=> , ET=> );
IF NOT In_EMG_RopeStop AND stFolder.Status.ApronBtmFold_AtHome  THEN
	IF NOT tonRopeStop.Q THEN
	Out_ClampUp:=TRUE;Out_ClampDown:=FALSE;
	_PumpA_SetVal	:=_PumpB_SetVal:=714;
	ELSE
		Out_ClampUp:=Out_ClampDown:=FALSE;
		_PumpA_SetVal	:=_PumpB_SetVal	:=0;
	END_IF
END_IF

//_PumpB_SetVal:=aa;



(**********************************************************************************************
******************	when first POWER ON , DualPump must run 50.0HZ last 5 minutes
******************	stFolder.PumpA_SetVal	:=iPumpA_SetVal;
******************	stFolder.PumpB_SetVal	:=iPumpB_SetVal;
***********************************************************************************************)
//IF GVL.FirstDualPump_5m THEN
//	_PumpA_SetVal	:=714;
//	_PumpB_SetVal	:=714;
//	Ton_Fst5Min(IN:= GVL.FirstDualPump_5m AND In_VltA_Running AND In_VltB_Running , PT:=T#1M);
//	IF Ton_Fst5Min.Q THEN
//		GVL.FirstDualPump_5m:=FALSE;
//	END_IF
//END_IF

fbPumpA(
	SetValue:=_PumpB_SetVal , 
	MinValue:=0 , 
	MaxValue:=1000 , 
	Options:=0 , 
	OUTPUT=>ANALOG_out_PumpA );
fbPumpB(
	SetValue:=_PumpA_SetVal , 
	MinValue:=0 , 
	MaxValue:=1000 , 
	Options:=0 , 
	OUTPUT=>ANALOG_out_PumpB );

//ANALOG_out_BtmApronSlide	:=REAL_TO_INT((LIMIT(-1000.0,rPropCmd_BtmSlide,1000.0)+1000.0)*32767.0/2000.0);
//ANALOG_out_BtmApronFold		:=REAL_TO_INT((LIMIT(-1000.0,rPropCmd_BtmFold,1000.0)+1000.0)*32767.0/2000.0);
//ANALOG_out_TopApronSlide	:=REAL_TO_INT((LIMIT(-1000.0,rPropCmd_TopSlide,1000.0)+1000.0)*32767.0/2000.0);
//ANALOG_out_TopApronFold		:=REAL_TO_INT((LIMIT(-1000.0,rPropCmd_TopFold,1000.0)+1000.0)*32767.0/2000.0);
IF Out_ApronTop_SlideFWD THEN
	ANALOG_out_TopApronSlide := 0;
ELSE
	ANALOG_out_TopApronSlide := REAL_TO_INT((LIMIT(-1430.0,rPropCmd_TopSlide,1430.0)+1430.0)*32767.0/2860.0);
END_IF

ANALOG_out_BtmApronSlide	:=REAL_TO_INT((LIMIT(-1430.0,rPropCmd_BtmSlide,1430.0)+1430.0)*32767.0/2860.0);
ANALOG_out_BtmApronFold		:=REAL_TO_INT((LIMIT(-1430.0,rPropCmd_BtmFold,1430.0)+1430.0)*32767.0/2860.0);
//ANALOG_out_TopApronSlide	:=REAL_TO_INT((LIMIT(-1430.0,rPropCmd_TopSlide,1430.0)+1430.0)*32767.0/2860.0);
ANALOG_out_TopApronFold		:=REAL_TO_INT((LIMIT(-1430.0,rPropCmd_TopFold,1430.0)+1430.0)*32767.0/2860.0);

IF rPropCmd_ClampUp >0 THEN
	ANALOG_out_ClampUp			:=REAL_TO_INT((LIMIT(-1000.0,rPropCmd_ClampUp,1000.0)+1000.0)*32767.0/2000.0);
	ANALOG_out_ClampDown		:=REAL_TO_INT((LIMIT(-1000.0,rPropCmd_ClampUp,1000.0)+1000.0)*32767.0/2000.0);
ELSIF rPropCmd_ClampDown >0 THEN
	ANALOG_out_ClampUp			:=REAL_TO_INT((LIMIT(-1000.0,rPropCmd_ClampDown,1000.0))*32767.0/2000.0);
	ANALOG_out_ClampDown		:=REAL_TO_INT((LIMIT(-1000.0,rPropCmd_ClampDown,1000.0))*32767.0/2000.0);
ELSE
	ANALOG_out_ClampUp			:=REAL_TO_INT((LIMIT(-1000.0,rPropCmd_ClampUp,1000.0)+1000.0)*32767.0/2000.0);
	ANALOG_out_ClampDown		:=REAL_TO_INT((LIMIT(-1000.0,rPropCmd_ClampUp,1000.0)+1000.0)*32767.0/2000.0);
END_IF

// Bypass proportional scaling for valve commissioning.
// Bipolar valves: idle = 12mA (midpoint), active = full 4mA/20mA.

//IF rPropCmd_BtmSlide > 0 THEN
//	ANALOG_out_BtmApronSlide	:=32767;
//ELSIF rPropCmd_BtmSlide < 0 THEN
//	ANALOG_out_BtmApronSlide	:=0;
//ELSE
//	ANALOG_out_BtmApronSlide	:=16384;
//END_IF

//IF rPropCmd_BtmFold > 0 THEN
//	ANALOG_out_BtmApronFold		:=32767;
//ELSIF rPropCmd_BtmFold < 0 THEN
//	ANALOG_out_BtmApronFold		:=0;
//ELSE
//	ANALOG_out_BtmApronFold		:=16384;
//END_IF

//IF rPropCmd_TopSlide > 0 THEN
//	ANALOG_out_TopApronSlide	:=32767;
//ELSIF rPropCmd_TopSlide < 0 THEN
//	ANALOG_out_TopApronSlide	:=0;
//ELSE
//	ANALOG_out_TopApronSlide	:=16384;
//END_IF

//IF rPropCmd_TopFold > 0 THEN
//	ANALOG_out_TopApronFold		:=32767;
//ELSIF rPropCmd_TopFold < 0 THEN
//	ANALOG_out_TopApronFold		:=0;
//ELSE
//	ANALOG_out_TopApronFold		:=16384;
//END_IF

//IF rPropCmd_ClampUp > 0 THEN
//	ANALOG_out_ClampUp			:=32767;
//	ANALOG_out_ClampDown		:=32767;
//ELSIF rPropCmd_ClampDown > 0 THEN
//	ANALOG_out_ClampDown		:=0;
//	ANALOG_out_ClampUp			:=0;
//ELSE
//	ANALOG_out_ClampUp			:=16384;
//	ANALOG_out_ClampDown		:=16384;
//END_IF



Out_PumpA_ST	:=In_PowerON;
//Out_PumpA_Rev	:=FALSE;
Out_PumpB_ST	:=In_PowerON;
//Out_PumpB_Rev	:=FALSE;

//************下滑动 下折弯 油缸意外滑动补偿 *开始******************/
tonSlipPatch_BtmSlide(IN:= NOT Out_ApronBtm_SlideFWD AND NOT Out_ApronBtm_SlideBWD AND NOT GVL.FirstDualPump_5m AND 
							stFolder.ApronBtm_Slide_ActPos<=6.0 AND stFolder.ApronBtm_Slide_ActPos>0.2 , PT:=T#1M , Q=> , ET=> );
//tonSlipPatch_BtmFold(IN:= NOT Out_ApronBtm_FoldFWD AND NOT Out_ApronBtm_FoldBWD AND NOT GVL.FirstDualPump_5m AND 
//							stFolder.ApronBtm_Fold_ActAngle<=9.0 AND stFolder.ApronBtm_Fold_ActAngle>0.2 , PT:=T#1M , Q=> , ET=> );
//bBtmSlide2:=NOT Out_ApronBtm_SlideFWD AND NOT Out_ApronBtm_SlideBWD AND 
//			stFolder.ApronBtm_Slide_ActPos<=6.0 AND stfolder.ApronBtm_Slide_ActPos<0.2 AND stfolder.ApronBtm_Slide_ActPos2>0.2;
IF tonSlipPatch_BtmSlide.Q OR bBtmSlide2 THEN
	gvl_bSlipPatch_BtmSlide	:=TRUE;
END_IF
//IF tonSlipPatch_BtmFold.Q THEN
//	gvl_bSlipPatch_BtmFold	:=TRUE;
//END_IF
tonSlipPatch_BtmSlidex(IN:=gvl_bSlipPatch_BtmSlide , PT:=T#2S , Q=> , ET=> );
//tonSlipPatch_BtmFoldx(IN:=gvl_bSlipPatch_BtmFold , PT:=T#2S , Q=> , ET=> );
IF tonSlipPatch_BtmSlidex.Q THEN
	gvl_bSlipPatch_BtmSlide	:=FALSE;
END_IF
//IF tonSlipPatch_BtmFoldx.Q THEN
//	gvl_bSlipPatch_BtmFold		:=FALSE;
//END_IF

//************下滑动 下折弯 油缸意外滑动补偿 *结束 ******************/

Out_PumpA_Load_Heav	:=	Out_ApronBtm_SlideFWD OR Out_ApronBtm_SlideBWD OR  Out_ApronBtm_FoldFWD OR Out_ApronBtm_FoldBWD 
						OR	Out_ClampUp OR
						(Out_ClampDown AND NOT stFolder.Status.Clamp_LtHalfPoint) OR
						(Out_ClampDown AND stFolder.Status.Clamp_LtHalfPoint AND SemiAuto_ActJob.ActType=1);
						
Out_PumpA_Load_Ligh	:=Out_ClampDown AND stFolder.Status.Clamp_LtHalfPoint AND SemiAuto_ActJob.ActType<>1 ;
						
Out_PumpB_Load_Heav	:=  Out_ApronTop_SlideFWD OR Out_ApronTop_SlideBWD OR Out_ApronTop_FoldFWD OR Out_ApronTop_FoldBWD
						OR Out_ClampUp 
						OR (Out_ClampDown AND NOT stFolder.Status.Clamp_LtHalfPoint)
						OR (Out_ClampDown AND stFolder.Status.Clamp_LtHalfPoint AND SemiAuto_ActJob.ActType=1)
//						OR Out_SlitterFwd OR Out_SlitterBwd 
						OR (Out_GaugingF_Ext OR Out_GaugingF_Rtn OR Out_GaugingR_Ext OR Out_GaugingR_Rtn);
						
Out_PumpB_Load_Ligh	:=Out_ClampDown AND stFolder.Status.Clamp_LtHalfPoint AND SemiAuto_ActJob.ActType<>1;





ftLoadRst(CLK:=Out_PumpA_Load_Ligh OR Out_PumpB_Load_Ligh OR Out_PumpA_Load_Heav OR Out_PumpB_Load_Heav, Q=> );
IF ftLoadRst.Q THEN
	stFolder.PumpA_SetVal	:=9;
	stFolder.PumpB_SetVal	:=9;
END_IF
END_ACTION

ACTION HMI:
Hmi_bArray[23]	:= NOT In_sigLaserFinger;  (*Turn OFF ,when Received Laser*)
Hmi_bArray[24]	:= In_sigClampMute;
Hmi_bArray[25]	:= stFolder.Status.Clamp_AtPressPoint;
Hmi_bArray[26]	:= (Operators>=1 AND (In_pedal1_UnClamp OR In_pedal1_Clamp OR In_pedal1_Slitter OR In_pedal1_SlitterBack
				OR In_pedal1_Fold OR In_pedal1_Gripper));


Hmi_bArray[30]	:= fbBackGauge.Axis_T1.ref.Status.Operational  AND fbBackGauge.Axis_T2.ref.Status.Operational 
					AND fbBackGauge.Axis_T3.ref.Status.Operational AND fbBackGauge.Axis_T4.ref.Status.Operational 
					AND fbBackGauge.Axis_Table.ref.Status.Operational;
Hmi_bArray[31]	:= fbBackGauge.Axis_T2.ref.Status.Coupled AND fbBackGauge.Axis_T3.ref.Status.Coupled AND fbBackGauge.Axis_T4.ref.Status.Coupled ;

Hmi_bArray[32]	:= In_sigTopApron_SlideFWD;
Hmi_bArray[33]	:= In_sigTopApron_FoldHome;
Hmi_bArray[34]	:= In_sigBtmApron_SlideFWD;
Hmi_bArray[35]	:= In_sigBtmApron_FoldHome;
Hmi_bArray[36]	:= In_sigLC_VLong;
Hmi_bArray[37]	:= In_sigLC_VShort;
Hmi_bArray[38]	:= In_sigLC_H;
Hmi_bArray[39]	:= NOT In_sigLaserFinger;

Hmi_bArray[100]	:=In_sigGaugingFrnt;
Hmi_bArray[101]	:=In_sigGaugingMid;
Hmi_bArray[102]	:=In_sigGaugingRear;

Hmi_bArray[104]	:=In_sigSlitLmt0;
Hmi_bArray[105]	:=In_sigSlitSlw0;
Hmi_bArray[106]	:=In_sigSlitLmt1;
Hmi_bArray[107]	:=In_sigSlitSlw1;

Hmi_iArray[20]	:= DINT_TO_UINT(fbUnitModeManager.eModeStatus);
Hmi_iArray[21]	:= Operators;

Hmi_rArray[20]	:=stFolder.ClampHt_ActPos;
Hmi_rArray[21]	:=stFolder.BackGauge_T1_ActPos+(stFolderPara.BackgaugeMaxPos-stFolderPara.MT1_BackstopZero);
Hmi_rArray[22]	:=stFolder.BackGauge_T2_ActPos+(stFolderPara.BackgaugeMaxPos-stFolderPara.MT2_BackstopZero);
Hmi_rArray[23]	:=stFolder.BackGauge_T3_ActPos+(stFolderPara.BackgaugeMaxPos-stFolderPara.MT3_BackstopZero);
Hmi_rArray[24]	:=stFolder.BackGauge_T4_ActPos+(stFolderPara.BackgaugeMaxPos-stFolderPara.MT4_BackstopZero);

Hmi_rArray[26]	:=stFolder.Table_ActPos;
Hmi_rArray[27]	:=stFolder.ApronTop_Slide_ActPos;
Hmi_rArray[28]	:=180-stFolder.ApronTop_Fold_ActAngle;
Hmi_rArray[29]	:=stFolder.ApronBtm_Slide_ActPos;
Hmi_rArray[30]	:=180-stFolder.ApronBtm_Fold_ActAngle;
Hmi_rArray[31]	:=0.0;		//Table Postion
Hmi_rArray[32]	:=stFolder.ClampPress;
Hmi_rArray[33]	:=ANALOG_in_PumpTemp*120.0/32767;			//Calibration value:  120.0--32767
Hmi_rArray[34]	:=ANALOG_out_PumpA*1500/32767;				//Calibration value:  1500.0--32767
Hmi_rArray[35]	:=ANALOG_out_PumpB*1500/32767;				//Calibration value:  1500.0--32767

Hmi_rArray[40]	:=stFolder.Feed_ActPos;

Hmi_bArray[103]	:=In_PumpLow_Alarm;

stFolderPara.bSemiAuto_Step			:=Hmi_bArray[61];
stFolderPara.bSemiAuto_Slitter		:=Hmi_bArray[62];
stFolderPara.bSemiAuto_BackGauge	:=Hmi_bArray[63];

stFolderPara.swSimplexDuplex		:=Hmi_bArray[0];
stFolderPara.swLightHeavy			:=Hmi_bArray[1];
stFolderPara.swSlitterVelocity		:=Hmi_bArray[2];
stFolderPara.swLoadingTable			:=Hmi_bArray[3];
stFolderPara.swAngleDisplay			:=Hmi_bArray[4];
stFolderPara.swClampOpen_InManual	:=Hmi_bArray[5];
stFolderPara.swClampOpen_InAuto		:=Hmi_bArray[6];
stFolderPara.swFeedMechanism		:=Hmi_bArray[7];

stFolderPara.SetFoldAngle		:=Hmi_rArray[50];
stFolderPara.SetMoveBackgauge	:=Hmi_rArray[51];
stFolderPara.SetTopApronSlide	:=Hmi_rArray[52];
stFolderPara.SetBtmApronSlide	:=Hmi_rArray[53];
stFolderPara.SetLoadingTable	:=Hmi_rArray[54];

stFolderPara.SetMoveFeed 		:=Hmi_rArray[57];


stFolderPara.Clamp_LowPos := Hmi_rArray[100];
stFolderPara.Clamp_MidPos := Hmi_rArray[101];
stFolderPara.Clamp_HighPos:=Hmi_rArray[102];
stFolderPara.Clamp_MaxPos:=Hmi_rArray[103];
stFolderPara.ClampHalfPos:=Hmi_rArray[104];
stFolderPara.Clamp_PressFlat:=Hmi_rArray[105];
stFolderPara.Clamp_FoldEnd:=Hmi_rArray[106];



stFolderPara.BackgaugeMaxPos:=Hmi_rArray[110];
stFolderPara.BackgaugeMinPos:=Hmi_rArray[111];
stFolderPara.SlitterOffset:=Hmi_rArray[112];
stFolderPara.BtmApronZeroPosition:=Hmi_rArray[113];
stFolderPara.TopApronZeroPosition:=Hmi_rArray[114];
stFolderPara.SquashBackstop_Top:=Hmi_rArray[115];
stFolderPara.SquashBackstop_Btm:=Hmi_rArray[116];
stFolderPara.SquashBackstop_External:=Hmi_rArray[117];
stFolderPara.SquashBackstop_OpenTop:=Hmi_rArray[118];
stFolderPara.SquashBackstop_OpenBtm:=Hmi_rArray[119];
stFolderPara.MT1_BackstopZero:=Hmi_rArray[120];
stFolderPara.MT2_BackstopZero:=Hmi_rArray[121];
stFolderPara.MT3_BackstopZero:=Hmi_rArray[122];
stFolderPara.MT4_BackstopZero:=Hmi_rArray[123];

FeedAuto_Job.Length			:=Hmi_iArray[90];
FeedAuto_Job.Width			:=Hmi_iArray[91];
FeedAuto_Job.Thickness		:=UINT_TO_REAL(Hmi_iArray[92])/10;
FeedAuto_Job.Quantity		:=Hmi_iArray[93];
FeedAuto_Job.Groups			:=Hmi_iArray[94];
FeedAuto_Job.Total			:=Hmi_iArray[95];
FeedAuto_Job.FeedPOS1		:=Hmi_rArray[90];
FeedAuto_Job.FeedPOS2		:=Hmi_rArray[91];

FeedDemoMode				:=Hmi_bArray[8];


stFolderPara.FeedOffset:=Hmi_rArray[107];
stFolderPara.FeedPosition:=Hmi_rArray[108];
stFolderPara.SetMoveFeed:=Hmi_rArray[109];
stFolderPara.Clamp_FeedPos	:=Hmi_rArray[94];

stFolderPara.BtmAngleAddit[iAdd]	:=Hmi_rArray[150+iAdd];
stFolderPara.TopAngleAddit[iAdd]	:=Hmi_rArray[170+iAdd];
iAdd:=(iAdd+1) MOD 15;
END_ACTION

{attribute 'object_name' := 'M_Execute'}
METHOD M_Execute
rtEnAuto(CLK:=fbUnitModeManager.eModeStatus=ePMLUnitMode_Auto , Q=> );
rtEnSemiAuto(CLK:=fbUnitModeManager.eModeStatus=ePMLUnitMode_SemiAuto , Q=> );
rtSlitterMode(CLK:=fbUnitModeManager.eModeStatus=ePMLUnitMode_AutoSlitter , Q=> );
CASE fbUnitModeManager.eModeStatus OF
	ePMLProtUnitMode_Production:		//Production
		A_SemiAuto();
	ePMLProtUnitMode_Maintenance:
		;
	ePMLUnitMode_Auto:
		A_SemiAuto();
		
	ePMLUnitMode_SemiAuto:	
		
		A_SemiAuto();
	ePMLUnitMode_AutoSlitter:
		A_SlitterAuto();
	ePMLProtUnitMode_Manual:		//Manual
		IF rtEnManual.Q THEN
			stFolderCom.TaskClamp	:=eTask_NULL;
			stFolderCom.TaskBackGauge	:=eTask_NULL;
			stFolderCom.TaskApron	:=eTask_NULL;
			stFolderCom.TaskSlitter	:=eTask_NULL;
			stFolderCom.TaskTable	:=eTask_NULL;
		END_IF
	
	
		
END_CASE
END_METHOD

METHOD M_SetUnitInfo
VAR_INPUT
END_VAR
aUnitInfo[eMachine].Name			:= 'fbMachine';
aUnitInfo[eMachine].ActMode		:= eMode;
aUnitInfo[eMachine].ActState		:= eState;

aUnitInfo[eUnit_Apron].Name			:= 'fbApron';
aUnitInfo[eUnit_Apron].ActMode		:= fbApron.eMode;
aUnitInfo[eUnit_Apron].ActState		:= fbApron.eState;

aUnitInfo[eUnit_BackGauge].Name			:= 'fbBackGuard';
aUnitInfo[eUnit_BackGauge].ActMode		:= fbBackGauge.eMode;
aUnitInfo[eUnit_BackGauge].ActState		:= fbBackGauge.eState;

aUnitInfo[eUnit_Clamp].Name		:= 'fbClamp';
aUnitInfo[eUnit_Clamp].ActMode	:= fbClamp.eMode;
aUnitInfo[eUnit_Clamp].ActState	:= fbClamp.eState;

aUnitInfo[eUnit_Slitter].Name		:= 'fbSlitter';
aUnitInfo[eUnit_Slitter].ActMode	:= fbSlitter.eMode;
aUnitInfo[eUnit_Slitter].ActState	:= fbSlitter.eState;
END_METHOD

END_FUNCTION_BLOCK

// ---- POUs/UNIT/fb_BackGauge/fb_BackGauge.TcPOU
FUNCTION_BLOCK fb_BackGauge EXTENDS FB_Generic
VAR_INPUT
		
	fbMasterClip:CYLINDER;
	fbT1_Clip:CYLINDER;
	fbT2_Clip:CYLINDER;
	fbT3_Clip:CYLINDER;
	bReset:BOOL;
	bAxisEnable:BOOL;
	
END_VAR
VAR_OUTPUT
END_VAR
VAR
	Axis_T1:Axis_PTPV3_CoE;
	Axis_T2:Axis_PTPV3_CoE;
	Axis_T3:Axis_PTPV3_CoE;
	Axis_T4:Axis_PTPV3_CoE;
	Axis_Table:Axis_PTPV3_CoE;
	Axis_Feed:Axis_PTPV3_CoE;
	
	i	:INT;
	s1	:BOOL;
	rtInGripper,rtInGripper2,rtInGripper3		:R_TRIG;
	iBackToZero: INT;
	fbBGAbsPos_T1,fbAbsPos_T2,fbAbsPos_T3,fbAbsPos_T4	:FB_BGAbsPos;
	fbTblAbsPos	:FB_TblAbsPos;
	fbFeedAbsPos:FB_FeedAbsPos;
	rtSuctionCup1,rtSuctionCup2:R_TRIG;
	AbsPos: INT;
	Task: INT;
	iBgStep: INT;
	iTableStep: INT;
	iGearStp: INT;
	iGearOutStp: INT;
	rtTemp1: R_trig;
	aa: BOOL;
	tonTemp1: TON;
	tonTemp2: Ton;
	GripAttach: REAL;
	in1,in2: INPUT;
	in3: INPUT;
	in4: INPUT;
	in_GearIn,in_GearOut: INPUT;
	ftReset: F_trig;
	tonOverTime1: Ton;
	tonOverTime2: Ton;
	tonOverTime3: Ton;
	TONGrip3 :Ton;
	
	TONSuctionCup1,TONSuctionCup2 :Ton;
	
	ix: INT;
	iZeroStp: INT;
	b1: BOOL;
	BGAbsRst: BOOL;
	RstDone: BOOL;
	tonRstDone: Ton;
	iBackBgStep: INT;
	iFeedStep: INT;

	TONFlipCup: Ton;
	tonTable: Ton;
END_VAR

SUPER^();
M01_Axis();
GearInOut();
stFolder.Status.Gripper	:=Out_Gripper;
stFolder.Status.Gripper2:=Out_Gripper2;
bReset	:=Hmi_bArray[41];

stFolder.Status.BG_Coupled	:= Axis_T2.ref.Status.Coupled AND Axis_T3.ref.Status.Coupled AND Axis_T4.ref.Status.Coupled;

IF fbUnitModeManager.eModeStatus=ePMLUnitMode_SemiAuto 
OR fbUnitModeManager.eModeStatus=ePMLUnitMode_AutoSlitter 
OR fbUnitModeManager.eModeStatus=ePMLUnitMode_Auto THEN
	CASE stFolderCom.paraBackGauge_GripType OF
	0:
		GripAttach	:=CNST_BACKGAUGE_ATTACH_PUSH;
		Out_GripperDatum_S0	:=FALSE;	Out_GripperDatum_S1:=FALSE;
	1:
		GripAttach	:=CNST_BACKGAUGE_ATTACH_GRIP;
		Out_GripperDatum_S0	:=FALSE;	Out_GripperDatum_S1:=FALSE;
	2:
		GripAttach	:=CNST_BACKGAUGE_ATTACH_OVERGRIP;
		Out_GripperDatum_S0	:=FALSE;	Out_GripperDatum_S1:=TRUE;
	4:
		GripAttach	:=CNST_BACKGAUGE_ATTACH_BACK;
		Out_GripperDatum_S0	:=TRUE;	Out_GripperDatum_S1:=FALSE;
	ELSE
		GripAttach	:=CNST_BACKGAUGE_ATTACH_PUSH;
		Out_GripperDatum_S0	:=TRUE;	Out_GripperDatum_S1:=TRUE;
	END_CASE
ELSIF fbUnitModeManager.eModeStatus=ePMLProtUnitMode_Manual THEN
	GripAttach	:=0;
	Out_GripperDatum_S0	:=FALSE;	Out_GripperDatum_S1:=FALSE;
END_IF

IF MAIN.fbMachine.bGripperDatumBack THEN
	Out_GripperDatum_S0	:=TRUE;	Out_GripperDatum_S1:=TRUE;
END_IF

TONGrip3(IN:=Out_Gripper3 , PT:=T#200MS , Q=> , ET=> );

IF fbUnitModeManager.eModeStatus=ePMLProtUnitMode_Manual
	OR fbUnitModeManager.eModeStatus=ePMLUnitMode_AutoSlitter
 	OR fbUnitModeManager.eModeStatus=ePMLUnitMode_SemiAuto
	OR fbUnitModeManager.eModeStatus=ePMLUnitMode_Auto THEN
	CASE stFolderCom.paraBackGauge_Grip OF
	0:
		Out_Gripper3:=TRUE;
		IF TONGrip3.Q THEN
			Out_Gripper:=TRUE;
			Out_Gripper2:=FALSE;
			stFolder.Status.GripperClose:=TRUE;
			stFolder.Status.GripperHalf:=stFolder.Status.GripperOpen:=FALSE;
		END_IF
	1:
		Out_Gripper:=Out_Gripper3:=FALSE;	
		Out_Gripper2	:=FALSE;
		stFolder.Status.GripperOpen:=TRUE;
		stFolder.Status.GripperClose:=stFolder.Status.GripperHalf:=FALSE;
//		IF  Axis_T1.ref.NcToPlc.ActPos >1120.0 OR ( stFolder.ClampHt_ActPos < 40 AND Axis_T1.ref.NcToPlc.ActPos >1020.0 ) THEN
//		Out_Gripper2:=TRUE;
//		stFolder.Status.GripperHalf:=TRUE;
//		stFolder.Status.GripperClose:=stFolder.Status.GripperOpen:=FALSE;
//		ELSE
//		Out_Gripper2	:=FALSE;
//		stFolder.Status.GripperOpen:=TRUE;
//		stFolder.Status.GripperClose:=stFolder.Status.GripperHalf:=FALSE;
//	 	END_IF
	END_CASE
END_IF


TONSuctionCup1(IN:=Out_SuctionCup1Suction OR Out_SuctionCup1Vent , PT:=T#2000MS , Q=> , ET=> );
IF fbUnitModeManager.eModeStatus=ePMLProtUnitMode_Manual
	OR fbUnitModeManager.eModeStatus=ePMLUnitMode_AutoFeed
 	OR fbUnitModeManager.eModeStatus=ePMLUnitMode_SemiAuto
	OR fbUnitModeManager.eModeStatus=ePMLUnitMode_Auto THEN
	CASE stFolderCom.paraFeed_SuctionCup1 OF	//1吸取 0释放
	1:
		Out_SuctionCup1Suction:= TRUE;
		IF TONSuctionCup1.Q THEN
			stFolder.Status.SuctionCup1:=TRUE;
		END_IF
	0:
		Out_SuctionCup1Suction:= FALSE;
		Out_SuctionCup1Vent	:=	stFolder.Status.SuctionCup1;
		IF TONSuctionCup1.Q THEN
			stFolder.Status.SuctionCup1:=FALSE;
		END_IF
	END_CASE
END_IF

TONSuctionCup2(IN:=Out_SuctionCup2Suction OR Out_SuctionCup2Vent , PT:=T#2000MS , Q=> , ET=> );
IF fbUnitModeManager.eModeStatus=ePMLProtUnitMode_Manual
	OR fbUnitModeManager.eModeStatus=ePMLUnitMode_AutoFeed
 	OR fbUnitModeManager.eModeStatus=ePMLUnitMode_SemiAuto
	OR fbUnitModeManager.eModeStatus=ePMLUnitMode_Auto THEN
	CASE stFolderCom.paraFeed_SuctionCup2 OF
	1:
		Out_SuctionCup2Suction:= TRUE;
		IF TONSuctionCup2.Q THEN
			stFolder.Status.SuctionCup2:=TRUE;
		END_IF
	0:
		Out_SuctionCup2Suction:= FALSE;
		Out_SuctionCup2Vent	:=	stFolder.Status.SuctionCup2;
		IF TONSuctionCup2.Q THEN
			stFolder.Status.SuctionCup2:=FALSE;
		END_IF
	END_CASE
END_IF


TONFlipCup(IN:=Out_FlipCupVent1 OR Out_FlipCupSuction1 , PT:=T#2000MS , Q=> , ET=> );
IF fbUnitModeManager.eModeStatus=ePMLProtUnitMode_Manual
	OR fbUnitModeManager.eModeStatus=ePMLUnitMode_AutoFeed
 	OR fbUnitModeManager.eModeStatus=ePMLUnitMode_SemiAuto
	OR fbUnitModeManager.eModeStatus=ePMLUnitMode_Auto THEN
	CASE stFolderCom.paraFlip_SuctionCup OF
	1:
		Out_FlipCupSuction1:= TRUE;
		Out_FlipCupSuction2:= TRUE;
		IF TONFlipCup.Q THEN
			stFolder.Status.FlipSuctionCup:=TRUE;
			TONFlipCup(IN:=FALSE);
		END_IF
	0:
		Out_FlipCupSuction1:= FALSE;
		Out_FlipCupSuction2:= FALSE;
		Out_FlipCupVent1	:=	stFolder.Status.FlipSuctionCup;
		Out_FlipCupVent2	:=	stFolder.Status.FlipSuctionCup;
		IF TONFlipCup.Q THEN
			stFolder.Status.FlipSuctionCup:=FALSE;
			TONFlipCup(IN:=FALSE);
		END_IF
	END_CASE
END_IF


IF stFolder.SlitterRef THEN
	stFolder.BackGauge_T1_ActPos:=stFolderPara.BackGaugeMaxPos + stFolderPara.SlitterOffset + GripAttach  - LREAL_TO_REAL(TRUNC(Axis_T1.ref.NcToPlc.ActPos*100))/100.0;
	stFolder.BackGauge_T2_ActPos:=stFolderPara.BackGaugeMaxPos + stFolderPara.SlitterOffset + GripAttach  - LREAL_TO_REAL(TRUNC(Axis_T2.ref.NcToPlc.ActPos*100))/100.0;
	stFolder.BackGauge_T3_ActPos:=stFolderPara.BackGaugeMaxPos + stFolderPara.SlitterOffset + GripAttach  - LREAL_TO_REAL(TRUNC(Axis_T3.ref.NcToPlc.ActPos*100))/100.0;
	stFolder.BackGauge_T4_ActPos:=stFolderPara.BackGaugeMaxPos + stFolderPara.SlitterOffset + GripAttach  - LREAL_TO_REAL(TRUNC(Axis_T4.ref.NcToPlc.ActPos*100))/100.0;
ELSE
	stFolder.BackGauge_T1_ActPos:=stFolderPara.BackGaugeMaxPos + GripAttach - LREAL_TO_REAL(TRUNC(Axis_T1.ref.NcToPlc.ActPos*100))/100.0;
	stFolder.BackGauge_T2_ActPos:=stFolderPara.BackGaugeMaxPos + GripAttach - LREAL_TO_REAL(TRUNC(Axis_T2.ref.NcToPlc.ActPos*100))/100.0;
	stFolder.BackGauge_T3_ActPos:=stFolderPara.BackGaugeMaxPos + GripAttach - LREAL_TO_REAL(TRUNC(Axis_T3.ref.NcToPlc.ActPos*100))/100.0;
	stFolder.BackGauge_T4_ActPos:=stFolderPara.BackGaugeMaxPos + GripAttach - LREAL_TO_REAL(TRUNC(Axis_T4.ref.NcToPlc.ActPos*100))/100.0;
END_IF
stFolder.BackGauge_T1_ActSpd:=LREAL_TO_REAL(TRUNC(Axis_T1.ref.NcToPlc.ActVelo*100))/100.0;
stFolder.BackGauge_T2_ActSpd:=LREAL_TO_REAL(TRUNC(Axis_T2.ref.NcToPlc.ActVelo*100))/100.0;
stFolder.BackGauge_T3_ActSpd:=LREAL_TO_REAL(TRUNC(Axis_T3.ref.NcToPlc.ActVelo*100))/100.0;
stFolder.BackGauge_T4_ActSpd:=LREAL_TO_REAL(TRUNC(Axis_T4.ref.NcToPlc.ActVelo*100))/100.0;
stFolder.Status.BackGauge_AtHome	:=(stFolder.BackGauge_T1_ActPos-stFolderPara.BackgaugeMaxPos)<CONST_BACKGAUGE_POS_Window;

stFolder.Table_ActPos:=LREAL_TO_REAL(TRUNC(Axis_Table.ref.NcToPlc.ActPos*100))/100.0;
stFolder.Table_ActSpd:=LREAL_TO_REAL(TRUNC(Axis_Table.ref.NcToPlc.ActVelo*100))/100.0;
stFolder.Status.Table_AtHome	:=stFolder.Table_ActPos<5.0;

stFolder.Feed_ActPos:=LREAL_TO_REAL(TRUNC(Axis_Feed.ref.NcToPlc.ActPos*100))/100.0;
stFolder.Feed_ActSpd:=LREAL_TO_REAL(TRUNC(Axis_Feed.ref.NcToPlc.ActVelo*100))/100.0;
stFolder.Status.Feed_AtHome	:=stFolder.Feed_ActPos>-100.0 AND stFolder.Feed_ActPos<5.0;
stFolder.Status.Feed_AtWork	:=stFolder.Feed_ActPos<-300.0;
GripperMan();


fbBGAbsPos_T1(
	Ex:= , 
	Mode:= , 
	Ax:=Axis_T1 , 
	TargetPos:=stFolderCom.paraBG_T1 , 
	ActPos:=stFolder.BackGauge_T1_ActPos,
	GripType:=stFolderCom.paraBackGauge_GripType , 
	GripOPEN:=stFolderCom.paraBackGauge_GripOPEN , 
	Velo:=stFolderCom.SpeedRatio_T1*stFolderCom.paraBackGaugeVelo ,
	Rst:=rtReset.Q , 
	RstDone	:=RstDone,
	Busy=> , 
	Done=> );
fbAbsPos_T2(
	Ex:= , 
	Mode:= , 
	Ax:=Axis_T2 , 
	TargetPos:=stFolderCom.paraBG_T2 , 	
	ActPos:=stFolder.BackGauge_T2_ActPos,
	GripType:=stFolderCom.paraBackGauge_GripType , 
	GripOPEN:=stFolderCom.paraBackGauge_GripOPEN , 
	Velo:=stFolderCom.SpeedRatio_T2*stFolderCom.paraBackGaugeVelo , 
	Rst:=rtReset.Q,
	RstDone	:=RstDone,
	Done=> );
fbAbsPos_T3(
	Ex:= , 
	Mode:= , 
	Ax:=Axis_T3 , 
	TargetPos:=stFolderCom.paraBG_T3 , 
	ActPos:=stFolder.BackGauge_T3_ActPos,
	GripType:=stFolderCom.paraBackGauge_GripType , 
	GripOPEN:=stFolderCom.paraBackGauge_GripOPEN , 
	Velo:=stFolderCom.SpeedRatio_T3*stFolderCom.paraBackGaugeVelo ,
	Rst:=rtReset.Q,
	RstDone	:=RstDone,
	Done=> );
fbAbsPos_T4(
	Ex:= , 
	Mode:= , 
	Ax:=Axis_T4 , 
	TargetPos:=stFolderCom.paraBG_T4 , 
	ActPos:=stFolder.BackGauge_T4_ActPos,
	GripType:=stFolderCom.paraBackGauge_GripType , 
	GripOPEN:=stFolderCom.paraBackGauge_GripOPEN , 
	Velo:=stFolderCom.SpeedRatio_T4*stFolderCom.paraBackGaugeVelo ,  
	Rst:=rtReset.Q,
	RstDone	:=RstDone,
	Done=> );
	
	
fbTblAbsPos(Ex:= , Ax:=Axis_Table , TargetPos:= ,Rst:=rtReset.Q, Done=> );
	
fbFeedAbsPos(Ex:= , Ax:=Axis_Feed , TargetPos:= ,Rst:=rtReset.Q, Done=> );

ACTION A_AutoRun:
(*
CASE i OF
	0:
	;
	1:
		Axis_T1.Motion.Velo:=CNST_BACKGAUGE_SPEED_HIGH;
		Axis_T1.Motion.Target:=200;
		Axis_T1.Motion.MoveAbs(TRUE);
		IF  Axis_T1.Motion.Done THEN
			i:=2;
			App.bBackStationPosFinish:=TRUE;
		END_IF
	2:
		
	IF 	App.bBendStationPosFinish  THEN
		i:=3;
	END_IF
	3:
		Axis_T1.NoAction();
		Axis_T2.NoAction();
		Axis_T3.NoAction();

		
	10:
		Axis_T2.Gear.RatioDenominator:=1;
		Axis_T2.Gear.RatioNumerator	:=1.0;
	//	Axis_T2.Gear.rMasterAxis1	:=Axis_T1.ref;
		Axis_T2.Gear.GearIn(TRUE);
		Axis_T3.Gear.RatioDenominator:=1;
		Axis_T3.Gear.RatioNumerator	:=1.0;
	//	Axis_T3.Gear.rMasterAxis1	:=Axis_T1.ref;
		Axis_T3.Gear.GearIn(TRUE);
	30:	
		Axis_T2.Gear.GearIn(FALSE);
		Axis_T3.Gear.GearIn(FALSE);
		
	40:
		Axis_T2.Gear.GearOut(TRUE);
		Axis_T3.Gear.GearOut(TRUE);
		41:
		Axis_T2.Gear.GearOut(FALSE);
		Axis_T3.Gear.GearOut(FALSE);
	20:
		M_StateComplete();
END_CASE
*)
END_ACTION

ACTION A_ManualRun:

(*Jog Control for All 4 Axis*)
	Axis_T1.Motion.Velo	:=CNST_BACKGAUGE_SPEED_HIGH;
	Axis_T1.HMI.JogPos		:= Hmi_bArray[110];
	Axis_T1.HMI.JogNeg 	:= Hmi_bArray[111];
	
//	Axis_Mx.Motion.Velo	:=CNST_BACKGAUGE_SPEED_HIGH;
//	Axis_Mx.HMI.JogPos 	:= Hmi_bArray[112];
//	Axis_Mx.HMI.JogNeg	:= Hmi_bArray[113];
		
	Axis_T2.Motion.Velo	:=CNST_BACKGAUGE_SPEED_HIGH;
	Axis_T2.HMI.JogPos 	:= Hmi_bArray[114];
	Axis_T2.HMI.JogNeg		:= Hmi_bArray[115];
		
	Axis_T3.Motion.Velo	:=CNST_BACKGAUGE_SPEED_HIGH;
	Axis_T3.HMI.JogPos 	:= Hmi_bArray[116];
	Axis_T3.HMI.JogNeg		:= Hmi_bArray[117];
		
	Axis_T4.Motion.Velo	:=CNST_BACKGAUGE_SPEED_HIGH;
	Axis_T4.HMI.JogPos 	:= Hmi_bArray[118];
	Axis_T4.HMI.JogNeg		:= Hmi_bArray[119];
	
	Axis_Table.Motion.Velo	:=CNST_TABLE_SPEED_HIGH;
	Axis_Table.HMI.JogPos 	:= Hmi_bArray[120];
	Axis_Table.HMI.JogNeg	:= Hmi_bArray[121];
	
	Axis_Feed.Motion.Velo	:=CONST_Feed_SPEED_LOW;
	Axis_Feed.HMI.JogPos 	:= Hmi_bArray[130];
	Axis_Feed.HMI.JogNeg	:= Hmi_bArray[131];
	
(*超时保护*)
tonOverTime1(IN:=Axis_T1.Motion.Busy , PT:=T#7S , Q=> , ET=> );
IF tonOverTime1.Q OR rtReset.Q THEN
	Axis_T1.NoAction();
	iBgStep	:=0;
	iBackToZero:=0;
END_IF

IF rtReset.Q THEN
	iBgStep	:=0;iBackToZero:=0;
	Axis_T1.Motion.MoveAbs(FALSE);
	Axis_T1.NoAction();
END_IF

(*1___后挡块移到零点*)
CASE iBackToZero OF
	0:
		IF Hmi_bArray[42] AND stFolder.ClampHt_ActPos > stFolderPara.ClampHalfPos THEN
			iBackToZero:=1;
		END_IF
	1:
		IF NOT stFolder.Status.Gripper THEN
			stFolderCom.paraBackGauge_Grip := 0;
		END_IF;
		IF stFolder.Status.Gripper THEN
			iBackToZero:=2;
		END_IF
	2:
		Axis_T1.NoAction();
		iBackToZero:=3;
	3:
		iBackToZero:=10;
	10:
		Axis_T1.Motion.Velo:=CNST_BACKGAUGE_SPEED_HIGH;
		Axis_T1.Motion.Target:=CONST_BACKGAUGE_POS_NegPlus;
		Axis_T1.Motion.MoveAbs(TRUE);
		IF  Axis_T1.Motion.Done THEN
			iBackToZero:=11;
			stFolder.Status.BackGauge_AtHome	:=TRUE;
		END_IF
	11:
		Axis_T1.NoAction();
		iBackToZero:=20;
	20:
		Axis_T1.Motion.Velo:=CNST_BACKGAUGE_SPEED_HIGH;
		Axis_T1.Motion.Target:=CONST_BACKGAUGE_POS_ZERO;
		Axis_T1.Motion.MoveAbs(TRUE);
		IF  Axis_T1.Motion.Done THEN
			iBackToZero:=21;
			stFolder.Status.BackGauge_AtHome	:=TRUE;
		END_IF
	21:
	IF 	stFolder.Status.BackGauge_AtHome  THEN
		iBackToZero:=0;
	END_IF
		
END_CASE

(*2___后挡块定位*)
CASE iBgStep OF
	0:
		IF Hmi_bArray[47] AND stFolder.ClampHt_ActPos > stFolderPara.ClampHalfPos THEN
			iBgStep	:=1;
			Axis_T1.NoAction();
		END_IF
	1:
		IF NOT stFolder.Status.Gripper THEN
			stFolderCom.paraBackGauge_Grip := 0;
		END_IF
		
		IF Hmi_rArray[51]>stFolder.BackGauge_T1_ActPos THEN
			iBgStep:=10;
		ELSE
			iBgStep:=20;
		END_IF
		
	10:
		Axis_T1.Motion.Velo:=CNST_BACKGAUGE_SPEED_HIGH;
		IF Hmi_bArray[46] THEN
			Axis_T1.Motion.Target:= LIMIT(-20, stFolderPara.BackGaugeMaxPos + stFolderPara.SlitterOffset - Hmi_rArray[51]-20,1210);
		ELSE
			Axis_T1.Motion.Target:= LIMIT(-20, stFolderPara.BackGaugeMaxPos - Hmi_rArray[51]-20,1210);
		END_IF;
		Axis_T1.Motion.MoveAbs(TRUE);
		IF  Axis_T1.Motion.Done THEN
			iBgStep:=11;
			stFolder.Status.BackGauge_AtHome	:=TRUE;
		END_IF
	11:
		Axis_T1.NoAction();
		iBgStep:=20;
	20:
		Axis_T1.Motion.Velo:=CNST_BACKGAUGE_SPEED_HIGH;
		IF Hmi_bArray[46] THEN
			Axis_T1.Motion.Target:= LIMIT(-20, stFolderPara.BackGaugeMaxPos + stFolderPara.SlitterOffset - Hmi_rArray[51],1210);
		ELSE
			Axis_T1.Motion.Target:= LIMIT(-20, stFolderPara.BackGaugeMaxPos - Hmi_rArray[51],1210);
		END_IF;
		iBgStep:=21;
	21:
		iBgStep:=22;
	22:
		iBgStep:=23;
	23:
		Axis_T1.Motion.MoveAbs(TRUE);
		IF  Axis_T1.Motion.Done THEN
			Axis_T1.NoAction();
			iBgStep:=30;
		END_IF
	30:
		Axis_T1.NoAction();
		iBgStep	:=0;
END_CASE;

tonOverTime2(IN:=Axis_Table.Motion.Busy , PT:=T#6.5S , Q=> , ET=> );
IF tonOverTime2.Q OR rtReset.Q THEN
	Axis_Table.NoAction();
	iTableStep	:=0;
END_IF
(*3___桌板定位*)
CASE iTableStep OF
	0:
		IF Hmi_bArray[51] AND stFolder.ClampHt_ActPos > stFolderPara.ClampHalfPos THEN
			iTableStep	:=1;
		END_IF
	1:
		Axis_Table.NoAction();
		iTableStep	:=2;
	2:
		iTableStep	:=3;
	3:
		iTableStep	:=4;
	4:
		iTableStep	:=5;
	5:
		Axis_Table.Motion.Velo:=CNST_TABLE_SPEED_HIGH;
		Axis_Table.Motion.Target:=LIMIT (CNST_TABLE_POS_MIN, Hmi_rArray[54], CNST_TABLE_POS_MAX);
		Axis_Table.Motion.MoveAbs(TRUE);
		IF  Axis_Table.Motion.Done THEN
			Axis_Table.NoAction();
			iTableStep	:=6;
		END_IF
	6:
		Axis_Table.NoAction();
		iTableStep	:=0;
END_CASE;


tonOverTime3(IN:=Axis_Feed.Motion.Busy , PT:=T#6.5S , Q=> , ET=> );
IF tonOverTime3.Q OR rtReset.Q THEN
	Axis_Feed.NoAction();
	iFeedStep	:=0;
END_IF
(*4___进料定位*)
CASE iFeedStep OF
	0:
		IF Hmi_bArray[54] AND stFolder.ClampHt_ActPos > stFolderPara.ClampHalfPos THEN
			iFeedStep	:=1;
		END_IF
	1:
		Axis_Feed.NoAction();
		iFeedStep	:=2;
	2:
		iFeedStep	:=3;
	3:
		iFeedStep	:=4;
	4:
		iFeedStep	:=5;
	5:
		Axis_Feed.Motion.Velo:=CONST_Feed_SPEED_HIGH;
		Axis_Feed.Motion.Target:=LIMIT (CONST_Feed_POS_MIN, Hmi_rArray[57], CONST_Feed_POS_MAX);
		Axis_Feed.Motion.MoveAbs(TRUE);
		IF  Axis_Feed.Motion.Done THEN
			Axis_Feed.NoAction();
			iFeedStep	:=6;
		END_IF
	6:
		Axis_Feed.NoAction();
		iFeedStep	:=0;
END_CASE;
END_ACTION

ACTION A_SemiAuto:
tonTemp1(IN:=stFolderCom.TaskBackGauge = eTask_BackGauge_AbsPos , PT:=T#100MS , Q=> , ET=> );
tonTemp2(IN:=stFolderCom.TaskBackGauge = eTask_BackGauge_BackPos , PT:=T#100MS , Q=> , ET=> );

in1(TrigDly_In:=stFolderCom.TaskBackGauge = eTask_BackGauge_AbsPos );
in2(TrigDly_In:=stFolderCom.TaskBackGauge = eTask_BackGauge_BackPos );
in_GearIn(TrigDly_In:=stFolderCom.TaskBackGauge = eTask_BackGauge_GearIn );
(*
in_GearOut(TrigDly_In:=stFolderCom.TaskBackGauge = eTask_BackGauge_GearOut );
*)
tonRstDone(IN:=RstDone , PT:=T#200MS , Q=> , ET=> );
IF tonRstDone.Q THEN
	RstDone:=FALSE;
END_IF
b1:=(fbUnitModeManager.eModeStatus=ePMLUnitMode_SemiAuto OR fbUnitModeManager.eModeStatus=ePMLUnitMode_Auto);
IF stFolderCom.TaskBackGauge = eTask_BackGauge_AbsPos THEN
	RstDone:=FALSE;
	fbBGAbsPos_T1.Ex		:=in1.TrigDly_Out;
	fbBGAbsPos_T1.Mode		:=1;	
	fbAbsPos_T2.Ex		:=fbAbsPos_T3.Ex	:=fbAbsPos_T4.Ex 	:=(b1 AND  stFolder.Taper_SW)	AND in1.TrigDly_Out;
	fbAbsPos_T2.Mode	:=fbAbsPos_T3.Mode	:=fbAbsPos_T4.Mode	:=1;
	IF (NOT (b1 AND stFolder.Taper_SW) AND fbBGAbsPos_T1.Done) OR
		((b1 AND stFolder.Taper_SW) AND fbBGAbsPos_T1.Done AND fbAbsPos_T2.Done 
						AND fbAbsPos_T3.Done AND fbAbsPos_T4.Done ) THEN
		
		stFolderCom.TaskBackGauge := eTask_NULL;
		RstDone:=TRUE;
		//fbBGAbsPos_T1.Ex	:=FALSE;
	END_IF
ELSIF stFolderCom.TaskBackGauge = eTask_BackGauge_BackPos  THEN
	RstDone:=FALSE;
	fbBGAbsPos_T1.Ex		:=in2.TrigDly_Out;
	fbBGAbsPos_T1.Mode		:=2;	
	fbAbsPos_T2.Ex		:=fbAbsPos_T3.Ex	:=fbAbsPos_T4.Ex	:=(b1 AND stFolder.Taper_SW) AND in2.TrigDly_Out;
	fbAbsPos_T2.Mode	:=fbAbsPos_T3.Mode	:=fbAbsPos_T4.Mode	:=2;
	IF (NOT (b1 AND stFolder.Taper_SW) AND fbBGAbsPos_T1.Done) OR
		((b1 AND stFolder.Taper_SW) AND fbBGAbsPos_T1.Done AND fbAbsPos_T2.Done 
						AND fbAbsPos_T3.Done AND fbAbsPos_T4.Done ) THEN
		stFolderCom.TaskBackGauge := eTask_NULL;
		RstDone:=TRUE;	
		fbBGAbsPos_T1.Ex	:=FALSE;
	END_IF
ELSIF stFolderCom.TaskBackGauge = eTask_BackGauge_GearIn THEN
	IF Axis_T2.ref.Status.Coupled AND Axis_T3.ref.Status.Coupled AND Axis_T4.ref.Status.Coupled THEN
		stFolderCom.TaskBackGauge := eTask_NULL;
	ELSE
		;
	END_IF
	(*
ELSIF stFolderCom.TaskBackGauge = eTask_BackGauge_GearOut THEN
	IF NOT Axis_T2.ref.Status.Coupled AND NOT Axis_T3.ref.Status.Coupled AND NOT Axis_T4.ref.Status.Coupled THEN
		stFolderCom.TaskBackGauge := eTask_NULL;
	ELSE
		;
	END_IF
	*)
ELSIF stFolderCom.TaskBackGauge = eTask_NULL THEN
	fbBGAbsPos_T1.Ex	:=FALSE;
	;
END_IF;

tonTable(IN:=stFolderCom.TaskTable = eTask_Table_AbsPos, PT:=T#200MS , Q=> , ET=> );

in3(TrigDly_In:=stFolderCom.TaskTable = eTask_Table_AbsPos);
IF stFolderCom.TaskTable = eTask_Table_AbsPos THEN
	fbTblAbsPos.Ex	:= in3.TrigDly_Out;
	fbTblAbsPos.TargetPos	:=stFolderCom.paraTablePos;
	IF fbTblAbsPos.Done THEN
		stFolderCom.TaskTable := eTask_NULL;
//		tonTable(IN:=FALSE);
	END_IF
END_IF;

in4(TrigDly_In:=stFolderCom.TaskFeed = eTask_Feed_AbsPos);
IF stFolderCom.TaskFeed = eTask_Feed_AbsPos THEN
	fbFeedAbsPos.Ex	:= in4.TrigDly_Out;
	fbFeedAbsPos.TargetPos	:=stFolderCom.paraFeedPos;
	IF fbFeedAbsPos.Done THEN
		stFolderCom.TaskFeed := eTask_NULL;
	END_IF
END_IF;
END_ACTION

ACTION GearInOut:
	ftReset(CLK:=bReset , Q=> );
IF ftReset.Q 
	OR in_GearIn.TrigDly_Out THEN
		iGearStp:=0;
	END_IF
IF in_GearOut.Q AND FALSE THEN
	iGearOutStp	:=10;
END_IF

(*Gear Ax ************************************************)
	CASE iGearStp OF
	0:
		IF Axis_T1.ref.Status.Operational  AND Axis_T2.ref.Status.Operational AND Axis_T3.ref.Status.Operational AND Axis_T4.ref.Status.Operational THEN
			iGearStp:=10;
		END_IF; 
	10:
		Axis_T2.Gear.GearOut(TRUE);
		Axis_T3.Gear.GearOut(TRUE);
		Axis_T4.Gear.GearOut(TRUE);
		iGearStp:=11;
	11:
		iGearStp:=12;
	12:
		iGearStp:=13;
	13:
		Axis_T2.Gear.GearOut(FALSE);
		Axis_T3.Gear.GearOut(FALSE);
		Axis_T4.Gear.GearOut(FALSE);
		iGearStp:=20;
		
	20:		//Abs Position
		Axis_T2.Motion.Velo:=CNST_BACKGAUGE_SPEED_HIGH;
		Axis_T2.Motion.Target:= Axis_T1.ref.NcToPlc.SetPos-10.0;
		Axis_T2.Motion.MoveAbs(TRUE);
		Axis_T3.Motion.Velo:=CNST_BACKGAUGE_SPEED_HIGH;
		Axis_T3.Motion.Target:= Axis_T1.ref.NcToPlc.SetPos-10.0;
		Axis_T3.Motion.MoveAbs(TRUE);
		Axis_T4.Motion.Velo:=CNST_BACKGAUGE_SPEED_HIGH;
		Axis_T4.Motion.Target:= Axis_T1.ref.NcToPlc.SetPos-10.0;
		Axis_T4.Motion.MoveAbs(TRUE);
		IF  Axis_T2.Motion.Done AND Axis_T3.Motion.Done AND Axis_T4.Motion.Done THEN
			iGearStp:=21;
		END_IF
	21:
		Axis_T2.NoAction();Axis_T3.NoAction();Axis_T4.NoAction();
		iGearStp:=30;
	30:

		Axis_T2.Motion.Target:= Axis_T1.ref.NcToPlc.SetPos+(stFolderPara.MT1_BackstopZero-stFolderPara.MT2_BackstopZero);
		Axis_T2.Motion.MoveAbs(TRUE);
		Axis_T3.Motion.Target:= Axis_T1.ref.NcToPlc.SetPos+(stFolderPara.MT1_BackstopZero-stFolderPara.MT3_BackstopZero);
		Axis_T3.Motion.MoveAbs(TRUE);
		Axis_T4.Motion.Target:= Axis_T1.ref.NcToPlc.SetPos+(stFolderPara.MT1_BackstopZero-stFolderPara.MT4_BackstopZero);
		Axis_T4.Motion.MoveAbs(TRUE);
		IF  Axis_T2.Motion.Done AND Axis_T3.Motion.Done AND Axis_T4.Motion.Done THEN
			iGearStp:=31;
		END_IF
	31:
		Axis_T2.NoAction();Axis_T3.NoAction();Axis_T4.NoAction();
		iGearStp:=40;
	40:		//Coupling Slave Axis
		Axis_T2.Gear.RatioDenominator:=1;
		Axis_T2.Gear.RatioNumerator	:=1.0;
		Axis_T2.Gear.GearIn(TRUE);
		Axis_T3.Gear.RatioDenominator:=1;
		Axis_T3.Gear.RatioNumerator	:=1.0;
		Axis_T3.Gear.GearIn(TRUE);
		Axis_T4.Gear.RatioDenominator:=1;
		Axis_T4.Gear.RatioNumerator	:=1.0;
		Axis_T4.Gear.GearIn(TRUE);
		iGearStp:=41;
	41:	
		Axis_T2.Gear.GearIn(FALSE);
		Axis_T3.Gear.GearIn(FALSE);
		Axis_T4.Gear.GearIn(FALSE);
		iGearStp:=50;
	50:
		IF  Axis_T2.ref.Status.Coupled AND Axis_T3.ref.Status.Coupled AND Axis_T4.ref.Status.Coupled THEN
			iGearStp:=100;
		ELSE
			iGearStp:=999;
		END_IF;
	100:
		;
	END_CASE

CASE iGearOutStp OF
	0:
		;
	10:
		Axis_T2.Gear.GearOut(TRUE);
		Axis_T3.Gear.GearOut(TRUE);
		Axis_T4.Gear.GearOut(TRUE);
		iGearOutStp:=11;
	11:
		Axis_T2.Gear.GearOut(FALSE);
		Axis_T3.Gear.GearOut(FALSE);
		Axis_T4.Gear.GearOut(FALSE);
		iGearOutStp:=100;
	
END_CASE
(*Back To Zero ************************************************)
CASE iZeroStp OF
	0:
		IF Hmi_bArray[11] THEN
			iZeroStp:=10;
		END_IF; 
	10:
		Axis_T2.Gear.GearOut(TRUE);
		Axis_T3.Gear.GearOut(TRUE);
		Axis_T4.Gear.GearOut(TRUE);
		iZeroStp:=11;
	11:
		iZeroStp:=12;
	12:
		iZeroStp:=13;
	13:
		Axis_T2.Gear.GearOut(FALSE);
		Axis_T3.Gear.GearOut(FALSE);
		Axis_T4.Gear.GearOut(FALSE);
		iZeroStp:=20;
	20:		//Abs Position
		Axis_T1.Motion.Velo:=CNST_BACKGAUGE_SPEED_HIGH;
		Axis_T1.Motion.Target:= 0-10.0;
		Axis_T1.Motion.MoveAbs(TRUE);
		Axis_T2.Motion.Velo:=CNST_BACKGAUGE_SPEED_HIGH;
		Axis_T2.Motion.Target:= 0-10.0;
		Axis_T2.Motion.MoveAbs(TRUE);
		Axis_T3.Motion.Velo:=CNST_BACKGAUGE_SPEED_HIGH;
		Axis_T3.Motion.Target:= 0-10.0;
		Axis_T3.Motion.MoveAbs(TRUE);
		Axis_T4.Motion.Velo:=CNST_BACKGAUGE_SPEED_HIGH;
		Axis_T4.Motion.Target:= 0-10.0;
		Axis_T4.Motion.MoveAbs(TRUE);
		IF Axis_T1.Motion.Done AND Axis_T2.Motion.Done AND Axis_T3.Motion.Done AND Axis_T4.Motion.Done THEN
			iZeroStp:=21;
		END_IF
	21:
		Axis_T1.NoAction(); Axis_T2.NoAction();Axis_T3.NoAction();Axis_T4.NoAction();
		iZeroStp:=30;
	30:
		Axis_T1.Motion.Target:= 0.0;
		Axis_T1.Motion.MoveAbs(TRUE);
		Axis_T2.Motion.Target:= 0.0;
		Axis_T2.Motion.MoveAbs(TRUE);
		Axis_T3.Motion.Target:= 0.0;
		Axis_T3.Motion.MoveAbs(TRUE);
		Axis_T4.Motion.Target:= 0.0;
		Axis_T4.Motion.MoveAbs(TRUE);
		IF Axis_T1.Motion.Done AND  Axis_T2.Motion.Done AND Axis_T3.Motion.Done AND Axis_T4.Motion.Done THEN
			iZeroStp:=31;
		END_IF
	31:
		Axis_T1.NoAction(); Axis_T2.NoAction();Axis_T3.NoAction();Axis_T4.NoAction();
		iZeroStp:=100;
	100:
		iZeroStp:=0;
END_CASE
END_ACTION

METHOD GripperMan
VAR_INPUT
END_VAR
(*rtInGripper(CLK:=pedal_Gripper , Q=> );
IF rtInGripper.Q AND stFolder.Status.Gripper THEN
	Out_Gripper	:=FALSE;
ELSIF rtInGripper.Q AND NOT stFolder.Status.Gripper THEN
	Out_Gripper	:=TRUE;
END_IF
*)

rtInGripper(CLK:=(In_pedal1_Gripper) , Q=> );

CASE Operators OF
	1:
		IF rtInGripper.Q AND stFolder.Status.Gripper THEN//开	
			stFolderCom.paraBackGauge_Grip := 1;
			stFolderCom.paraBackGauge_GripOPEN := TRUE;
		ELSIF rtInGripper.Q AND NOT stFolder.Status.Gripper THEN//夹紧
			stFolderCom.paraBackGauge_Grip := 0;	
			stFolderCom.paraBackGauge_GripOPEN := FALSE;
		END_IF
	2,3,4:
		IF rtInGripper.Q AND stFolder.Status.Gripper THEN
			Out_Gripper	:=FALSE;
		ELSIF rtInGripper.Q AND NOT stFolder.Status.Gripper THEN
			Out_Gripper	:=TRUE;
		END_IF
		IF rtInGripper2.Q AND stFolder.Status.Gripper2 THEN
			Out_Gripper2	:=FALSE;
		ELSIF rtInGripper2.Q AND NOT stFolder.Status.Gripper2 THEN
			Out_Gripper2	:=TRUE;
		END_IF
END_CASE

rtInGripper3(CLK:=(Hmi_bArray[87]) , Q=> );

IF rtInGripper3.Q AND GripAttach = CNST_BACKGAUGE_ATTACH_BACK THEN 
	stFolderCom.paraBackGauge_GripType := 1;
ELSIF rtInGripper3.Q AND GripAttach = CNST_BACKGAUGE_ATTACH_GRIP THEN 
	stFolderCom.paraBackGauge_GripType := 2;
ELSIF rtInGripper3.Q AND GripAttach = CNST_BACKGAUGE_ATTACH_OVERGRIP THEN 
	stFolderCom.paraBackGauge_GripType := 4;
END_IF

IF fbUnitModeManager.eModeStatus=ePMLProtUnitMode_Manual THEN
	stFolderCom.paraFeed_SuctionCup1:=BOOL_TO_INT(Hmi_bArray[55]);
	stFolderCom.paraFeed_SuctionCup2:=BOOL_TO_INT(Hmi_bArray[56]);
END_IF


IF fbUnitModeManager.eModeStatus=ePMLProtUnitMode_Manual THEN
	stFolderCom.paraFlip_SuctionCup:=BOOL_TO_INT(Hmi_bArray[57]);
END_IF
END_METHOD

{attribute 'object_name' := 'M_Execute'}
METHOD M_Execute
VAR
	



END_VAR

CASE fbUnitModeManager.eModeStatus OF
	ePMLProtUnitMode_Production:		//Production
		;
	ePMLProtUnitMode_Maintenance:		
		//
		;
	ePMLUnitMode_Auto:
		A_SemiAuto();
	ePMLUnitMode_SemiAuto:
		A_SemiAuto();
	ePMLUnitMode_AutoSlitter:
		A_SemiAuto();
	ePMLProtUnitMode_Manual:		//Manual
		A_ManualRun();
	stFolder.SlitterRef:=Hmi_bArray[46];

		
 
		
		
END_CASE   
	
	//A_AutoRun();
END_METHOD

METHOD M01_Axis
VAR_INPUT
END_VAR

VAR
END_VAR
(* XAx *****************************************************************)
	Axis_T1.Admin.RST											:= bReset;
	Axis_T1.Admin.Enable 										:= (*Axis_T1.para.InitDone AND Axis_T1.drive.Ready AND *)bAxisEnable;
																														
	Axis_T1.Admin.EnableNeg 									:=TRUE;
	Axis_T1.Admin.EnablePos 									:= TRUE;
	Axis_T1.Admin.Override										:= 100;
	                                        		
	Axis_T1.HMI.Enable											:=eMode=ePMLProtUnitMode_Manual AND eState=ePMLState_Execute;
		                                    		
	Axis_T1.Home.Mode											:= MC_HomingMode.MC_DefaultHoming;
	(*
	Axis_T1.Home.Pos											;
	Axis_T1.Home.CalibrationCam									;
	Axis_T1.Home.AcceptBlockedDrive								;
	                                        		                                  	
	Axis_T1.Drive.ErrorEndlageNeg								;
	Axis_T1.Drive.ErrorEndlagePos								;	
	Axis_T1.Drive.EnableEvent								    ;
 	  *)                                     		       
	(* Call Axis *)                         		
	Axis_T1();                                  		
	
(* T1Ax *****************************************************************)
	Axis_T2.Admin.RST											:= bReset;
	Axis_T2.Admin.Enable 										:= (*Axis_T1.para.InitDone AND Axis_T1.drive.Ready AND*) bAxisEnable;
																														
	Axis_T2.Admin.EnableNeg 									:=TRUE;
	Axis_T2.Admin.EnablePos 									:= TRUE;
	Axis_T2.Admin.Override										:= 100;
	                                        		
	Axis_T2.HMI.Enable											:=eMode=ePMLProtUnitMode_Manual AND eState=ePMLState_Execute;
		                                    		
	Axis_T2.Home.Mode											:= MC_HomingMode.MC_DefaultHoming;
		(*
	Axis_T2.Home.Pos											;
	Axis_T2.Home.CalibrationCam									;
	Axis_T2.Home.AcceptBlockedDrive								;
	                                        		                                  	
	Axis_T2.Drive.ErrorEndlageNeg								;
	Axis_T2.Drive.ErrorEndlagePos								;	
	Axis_T2.Drive.EnableEvent								    ;
 	                 *)                       		       
	(* Call Axis *)                         		
	Axis_T2(rMasterAxis:=Axis_T1.ref);         

(* T2Ax *****************************************************************)

	Axis_T3.Admin.RST											:= bReset;
	Axis_T3.Admin.Enable 										:=(* Axis_T1.para.InitDone AND Axis_T1.drive.Ready AND*) bAxisEnable;
																														
	Axis_T3.Admin.EnableNeg 									:=TRUE;
	Axis_T3.Admin.EnablePos 									:= TRUE;
	Axis_T3.Admin.Override										:= 100;
	                                        		
	Axis_T3.HMI.Enable											:=eMode=ePMLProtUnitMode_Manual AND eState=ePMLState_Execute;
		                                    		
	Axis_T3.Home.Mode											:= MC_HomingMode.MC_DefaultHoming;
		(*
	Axis_T3.Home.Pos											;
	Axis_T3.Home.CalibrationCam									;
	Axis_T3.Home.AcceptBlockedDrive								;
	                                        		                                  	
	Axis_T3.Drive.ErrorEndlageNeg								;
	Axis_T3.Drive.ErrorEndlagePos								;	
	Axis_T3.Drive.EnableEvent								    ;
 	                    *)                    		       
	(* Call Axis *)                         		
	Axis_T3(rMasterAxis:=Axis_T1.ref);       
	
	
	(* T3Ax *****************************************************************)

	Axis_T4.Admin.RST											:= bReset;
	Axis_T4.Admin.Enable 										:= (*Axis_T1.para.InitDone AND Axis_T1.drive.Ready AND*) bAxisEnable;
																														
	Axis_T4.Admin.EnableNeg 									:=TRUE;
	Axis_T4.Admin.EnablePos 									:= TRUE;
	Axis_T4.Admin.Override										:= 100;
	                                        		
	Axis_T4.HMI.Enable											:=eMode=ePMLProtUnitMode_Manual AND eState=ePMLState_Execute;
		                                    		
	Axis_T4.Home.Mode											:= MC_HomingMode.MC_DefaultHoming;
		(*
	Axis_T4.Home.Pos											;
	Axis_T4.Home.CalibrationCam									;
	Axis_T4.Home.AcceptBlockedDrive								;
	                                        		                                  	
	Axis_T4.Drive.ErrorEndlageNeg								;
	Axis_T4.Drive.ErrorEndlagePos								;	
	Axis_T4.Drive.EnableEvent								    ;
 	          *)                              		       
	(* Call Axis *)                         		
	Axis_T4(rMasterAxis:=Axis_T1.ref);      

	
	(* Table Ax *****************************************************************)

	Axis_Table.Admin.RST											:= bReset;
	Axis_Table.Admin.Enable 										:= (*Axis_T1.para.InitDone AND Axis_T1.drive.Ready AND*) bAxisEnable;
																														
	Axis_Table.Admin.EnableNeg 									:=TRUE;
	Axis_Table.Admin.EnablePos 									:= TRUE;
	Axis_Table.Admin.Override										:= 100;
	                                        		
	Axis_Table.HMI.Enable											:=eMode=ePMLProtUnitMode_Manual AND eState=ePMLState_Execute;
		                                    		
	Axis_Table.Home.Mode											:= MC_HomingMode.MC_DefaultHoming;
		(*
	Axis_T4.Home.Pos											;
	Axis_T4.Home.CalibrationCam									;
	Axis_T4.Home.AcceptBlockedDrive								;
	                                        		                                  	
	Axis_T4.Drive.ErrorEndlageNeg								;
	Axis_T4.Drive.ErrorEndlagePos								;	
	Axis_T4.Drive.EnableEvent								    ;
 	          *)                              		       
	(* Call Axis *)                         
		
	Axis_Table(rMasterAxis:=Axis_Table.ref);     
 
	(* Feed Ax *****************************************************************)

	Axis_Feed.Admin.RST											:= bReset;
	Axis_Feed.Admin.Enable 										:= (*Axis_T1.para.InitDone AND Axis_T1.drive.Ready AND*) bAxisEnable;
																														
	Axis_Feed.Admin.EnableNeg 									:=TRUE;
	Axis_Feed.Admin.EnablePos 									:= TRUE;
	Axis_Feed.Admin.Override										:= 100;
	                                        		
	Axis_Feed.HMI.Enable											:=eMode=ePMLProtUnitMode_Manual AND eState=ePMLState_Execute;
		                                    		
	Axis_Feed.Home.Mode											:= MC_HomingMode.MC_DefaultHoming;
		(*
	Axis_T4.Home.Pos											;
	Axis_T4.Home.CalibrationCam									;
	Axis_T4.Home.AcceptBlockedDrive								;
	                                        		                                  	
	Axis_T4.Drive.ErrorEndlageNeg								;
	Axis_T4.Drive.ErrorEndlagePos								;	
	Axis_T4.Drive.EnableEvent								    ;
 	          *)                              		       
	(* Call Axis *)                         		
	Axis_Feed(rMasterAxis:=Axis_Feed.ref);
END_METHOD

END_FUNCTION_BLOCK

// ---- POUs/UNIT/fb_BackGauge/FB_FeedAbsPos.TcPOU
FUNCTION_BLOCK FB_FeedAbsPos
VAR_INPUT
	Ex			:BOOL;
	TargetPos	:LREAL;
	Rst	:BOOL;
END_VAR
VAR_OUTPUT
	Done	:BOOL;
END_VAR
VAR_IN_OUT
	Ax			:Axis_PTPV3_CoE;
END_VAR
VAR
	iPTP: INT;
	GripAttach	:REAL;
	ton1: Ton;
	ton2: Ton;
	rTemp0: REAL;
END_VAR

IF Rst THEN
	iPTP	:=100;
END_IF

CASE iPTP OF
	0:
	IF Ex THEN
		iPTP	:=1;
		Done:=FALSE;
	END_IF
	1:
		Ax.NoAction();
		iPTP	:=10;
	10:
		iPTP:=11;
	11:
		iPTP:=12;
	12:
		Ax.Motion.Velo:=stFolderCom.paraFeedVelo;
		Ax.Motion.Target:= LIMIT(CONST_FEED_POS_MIN, TargetPos,CONST_FEED_POS_MAX);
		Ax.Motion.MoveAbs(TRUE);
		IF  Ax.Motion.Done  OR ABS(Ax.Motion.Target-Ax.ref.NcToPlc.ActPos)<0.1 THEN
			iPTP:=100;
		END_IF
	100:
		Ax.Motion.MoveAbs(FALSE);
		iPTP:=101;
	101:
		Ax.NoAction();
		iPTP:=0;
		Done:=TRUE;

		
END_CASE

ton1(IN:=Done , PT:=T#1S , Q=> , ET=> );
IF ton1.Q THEN 
	Done:=FALSE;
END_IF

END_FUNCTION_BLOCK

// ---- POUs/UNIT/fb_Slitter/fb_Slitter.TcPOU
FUNCTION_BLOCK fb_Slitter EXTENDS FB_Generic
VAR_INPUT
END_VAR
VAR_OUTPUT
END_VAR
VAR
	iManSlitStep	:INT;
	rtPedalSlite	:R_TRIG;
	tonPedalSlite	:TON;
	bTmp1: BOOL;
	bManSlitRunning: BOOL;
	i: INT;
	fbSlitterAct	:FB_SlitterAct;
END_VAR

SUPER^();
//tonPedalSlite(IN:=In_pedal1_Slitter , PT:=T#2S , Q=> , ET=> );

stFolder.Status.Slitter_AtHome	:=In_sigSlitLmt0;

fbSlitterAct(Done=> );

Out_SlitterFwd	:=fbSlitterAct.bOutSlitterFwd AND In_sigBtmApron_SlideFWD AND In_sigBtmApron_FoldHome;
Out_SlitterBwd	:=fbSlitterAct.bOutSlitterBwd AND In_sigBtmApron_SlideFWD AND In_sigBtmApron_FoldHome;



IF NOT stFolder.Status.SlitterAtSlow AND NOT Hmi_bArray[88] AND NOT Hmi_bArray[89] THEN
	Out_SlitterSpeed:= TRUE;
ELSE
	Out_SlitterSpeed:= FALSE;
END_IF		

IF Hmi_bArray[88] THEN 
	Out_SlitterFwd := TRUE;
END_IF

IF Hmi_bArray[89] THEN 
	Out_SlitterBwd := TRUE;
END_IF

ACTION A_AutoRun:

END_ACTION

ACTION A_ManualRun:

END_ACTION

{attribute 'object_name' := 'M_Execute'}
METHOD M_Execute

VAR
	
END_VAR
CASE fbUnitModeManager.eModeStatus OF
	ePMLProtUnitMode_Production:		//Production
		;
		
	ePMLProtUnitMode_Maintenance:		
		//
		;
		ePMLUnitMode_Auto:
		IF stFolderCom.TaskSlitter =eTask_SlitterAct THEN
			IF fbSlitterAct.Done THEN
				stFolderCom.TaskSlitter	:=eTask_NULL;
			END_IF
		END_IF
	ePMLUnitMode_SemiAuto:
		i:=334;
		IF stFolderCom.TaskSlitter =eTask_SlitterAct THEN
			IF fbSlitterAct.Done THEN
				stFolderCom.TaskSlitter	:=eTask_NULL;
			END_IF
		END_IF
	ePMLUnitMode_AutoSlitter:
		i:=339;
		IF stFolderCom.TaskSlitter =eTask_SlitterAct THEN
			IF fbSlitterAct.Done THEN
				stFolderCom.TaskSlitter	:=eTask_NULL;
			END_IF
		END_IF
	ePMLProtUnitMode_Manual:		//Manual
		A_ManualRun();
		stFolderCom.TaskSlitter :=eTask_SlitterAct;


		//Out_SlitterFwd	:=In_pedal1_Slitter AND NOT In_sigSlitSlw1 AND NOT In_sigSlitLmt1 ;
		//Out_SlitterBwd	:=In_pedal1_SlitterBack;
		
		

		
END_CASE
END_METHOD

END_FUNCTION_BLOCK

// ---- POUs/PTP/01_Base/Ax_AdminCtrl.TcPOU
{attribute 'no_check'}
FUNCTION_BLOCK Ax_AdminCtrl (* axis reset, set operational, start and stop *)
VAR_INPUT
	RST														:	BOOL := FALSE; // Reset NC Error and restart current cmd if possible
	Enable													: 	BOOL := FALSE; // Cyclic NCAxis enable operational - FALSE = Stop 
	EnablePos												: 	BOOL := FALSE; // feed enable positiv 
	EnableNeg												: 	BOOL := FALSE; // Vorschubreigabe Negativ 
	BufferMode												:	MC_BufferMode := MC_Aborting;	(* 	MC_Aborting,
																									MC_Buffered,
																									MC_BlendingLow,
																									MC_BlendingPrevious,
																									MC_BlendingNext,
																									MC_BlendingHigh *) 
                                							
	Override												:	LREAL; // Override 
	rAxis													:	REFERENCE TO AXIS_REF := 0;
	ShowNCErrIfDisabled										:	BOOL := FALSE;
END_VAR                         							
VAR_IN_OUT                      							
END_VAR                         							
VAR_OUTPUT                      							
	EnableOK												:	BOOL; // Enable is send to NC
	Ready													:	BOOL;
	StartRel												:	BOOL;
	Busy													:	BOOL;
	Done													:	BOOL;
	Error													:	BOOL;
	ErrorID													:	UDINT;
	ErrorText												:	STRING(40);
END_VAR
VAR
(* Zwischenspeicher **************************************************************************)
	MethSeqEnable											: 	BOOL := TRUE;	(* NCAchse BTB/Freigabe setzen - FALSE = Stop, auch ueber Methoden set/reset bar *)
	                        	
(* Timer *)                 	
	TON_Ready												:	TON;

(* Trigger *)

(* Instanzierung der MC Bausteine *******************************************************)
	MC_Power												: MC_Power;
	MC_Reset												: MC_Reset;

(* Dummy Speicher **********************************************************)

(* Skalierungsfaktor ermitteln *********************************************
	Skalierungsfaktor von 0.1 eintragen. Istpositon "Anfang" merken.
	Antrieb um einen realen Wert "X" mm verfahren. Differenz der
	momentanen Istposition zur Istposition "Anfang" ermitteln.
	SKalierungsfaktor =		realer Fahrweg 
							---------------------------
							Differenz der Istpositionen
*)
END_VAR

	(************************************************************************************)
	(*																					*)
	(*		B E C K H O F F   N E W   A U T O M A T I O N   T E C H N O L O G Y    		*)
	(*																					*)
	(*		Eiserstr.5	D-33415 Verl	Germany	phone:	+49-5246-0	www.Beckhoff.Com	*)
    (*																					*)
    (*		Bausteinbeschreibung	:	Power/Reset Achs Baustein						*)
	(*		TwinCAT-Version			:	3.x or higher									*)
	(*		Version					:	V1.1 	 										*)
 	(*		Autor					:	DS												*)
	(*																					*)
	(*	call function-block cyclically for enableing axis and refresh REF.Status		*)
	(************************************************************************************)

(* abortinf function-block-call if reference is invalid *********************************)
IF NOT __ISVALIDREF(rAxis) THEN
	EnableOK												:= FALSE;
	Busy													:= NOT Error;
	Ready													:= FALSE;
	Error													:= TRUE;
	ErrorId													:= 16#4B30;
	Done													:= FALSE;
	StartRel												:= FALSE;
	ErrorText												:= 'Reference rAxis invalid (0)';
	RETURN;	
END_IF

(* rading axis-status from NCtoPLC-channel ***********************************************)
	rAxis.ReadStatus();

(* set axis operational  *****************************************************************)
	MC_Power(
		Enable			:= Enable AND MethSeqEnable,
		Enable_Positive	:= EnablePos,
		Enable_Negative	:= EnableNeg,
		Override		:= LIMIT(0.0,Override,100.0),
		BufferMode		:= (* PwrBufferMode *),
		Axis			:= rAxis,
		Status			=> ,
		Busy			=> ,
		Active			=> ,
		Error			=> ,
		ErrorID			=> );

(* Reset axis ****************************************************************)
	MC_Reset(
		Execute	:= 	RST 
					AND rAxis.Status.PTPmode 
					AND (rAxis.NcToPlc.ErrorCode <> 0 OR NOT rAxis.Status.HasJob)
					OR MC_Reset.Execute,
		Axis	:= rAxis,
		Done	=> Done,
		Busy	=> Busy,
		Error	=> ,
		ErrorID	=> );
		
	MC_Reset.Execute										:= FALSE; 	

(********************************************************************************)
(* axis status																	*)
(********************************************************************************)
	(* Axis Enabled *)
	EnableOK 												:= MC_Power.Enable;

	(* Axis Ready *)
	TON_Ready(
		IN := MC_Power.Status
				AND NOT rAxis.Status.DriveDeviceError
				AND NOT rAxis.Status.IoDataInvalid
				AND NOT rAxis.Status.Error
				AND NOT rAxis.Status.ErrorStop,
		PT 	:= T#50MS, (* 100ms BoschRex Sercos 2 *)
		Q	=> Ready);

	(* Axis Ready to Start *)
	StartRel												:= Ready
																AND rAxis.Status.PTPmode
																AND NOT rAxis.Status.ProtectedMode
																AND NOT rAxis.Status.MotionCommandsLocked
																AND (MC_Power.Enable_Negative OR MC_Power.Enable_Positive);
                                							
(******************************************************************************)
(* Ctrl Status 																					*)
(******************************************************************************)
	IF MC_Power.Error
		AND NOT MC_Reset.Execute
	THEN
		Error												:= TRUE;
		ErrorId												:= MC_Power.ErrorID;
		ErrorText											:= CONCAT('MC_Power ErrorId: ', UDINT_TO_STRING(Errorid));
	ELSIF MC_Reset.Execute  								
		AND MC_Reset.Error  								
	THEN                    								
		Error												:= TRUE;
		ErrorId												:= MC_Reset.ErrorID;
		ErrorText											:= CONCAT('MC_Reset ErrorId: ', UDINT_TO_STRING(Errorid));
	ELSIF rAxis.NcToPlc.ErrorCode <> 0 AND ShowNCErrIfDisabled
	THEN
		Error												:= TRUE;
		ErrorId												:= rAxis.NcToPlc.ErrorCode;
		ErrorText											:= CONCAT('NC ErrorId: ', UDINT_TO_STRING(Errorid));
	ELSE                    								
		Error													:= FALSE;
		ErrorId												:= 0;
		ErrorText											:= '';
	END_IF

(**************************************************************************************************)

METHOD PUBLIC ForceFeed : BOOL //Return = IN - Force Inputparameter 
VAR_INPUT
	IN														:	booL;
END_VAR
THIS^.EnableNeg 											:= IN;
THIS^.EnablePos 											:= IN;

ForceFeed 													:= IN;
END_METHOD

METHOD PUBLIC Reset : BOOL //Return = Busy
//required parameter
//rAxis
VAR_INPUT
	IN						:	BOOL;
END_VAR
IF NOT __ISVALIDREF(rAxis) 
THEN
	Busy													:= NOT Error;
	Error													:= TRUE;
	ErrorId													:= 16#4B30;
	Done													:= FALSE;
	ErrorText												:= 'Reference rAxis invalid (0)';
	RETURN;             								
END_IF

	MC_Reset(
		Execute	:= NOT rAxis.Status.ProtectedMode
						AND (		RST 
								OR IN 
								OR rAxis.NcToPlc.ErrorCode <> 0 
								OR NOT rAxis.Status.HasJob) ,
		Axis	:= rAxis,
		Done	=> Done,
		Busy	=> Busy,
		Error	=> Error,
		ErrorID	=> ErrorId);

	IF Error 
	THEN
		ErrorText											:= SEL(MC_Reset.Error , '' ,  CONCAT('Error MC_Reset id: ',  UDINT_TO_STRING(Errorid)));
	ELSE            										
		ErrorText											:= '';
	END_IF          										
	                	
	Reset													:= Busy;
END_METHOD

METHOD PUBLIC SeqEnable : BOOL //Return = Ready - Enable and disabel per method from external
VAR_INPUT
IN															:	BOOL;
END_VAR
THIS^.MethSeqEnable 										:= IN;
SeqEnable													:= Ready;
END_METHOD

END_FUNCTION_BLOCK

// ---- POUs/PTP/03_Utilities/GetAxErrTxt.TcPOU
{attribute 'no_check'}
FUNCTION GetAxErrTxt : STRING
VAR_INPUT
	Quelle													:	STRING(20);
	ErrorID													:	DINT;
END_VAR         											
VAR
END_VAR

	(************************************************************************************)
	(*																					*)
	(*		B E C K H O F F   N E W   A U T O M A T I O N   T E C H N O L O G Y    		*)
	(*																					*)
	(*		Eiserstr.5	D-33415 Verl	Germany	phone:	+49-5246-0	www.Beckhoff.Com	*)
    (*																					*)
    (*		Bausteinbeschreibung	:	Gibt einen Infotext zur angegebenen ErrorID aus,*)
	(*										hinterlegt sind Achs und ADS Errorids		*)
	(*		Version					:	V1.1 / 09/07									*)
	(*																					*)
	(************************************************************************************)


(* Work info Txt ***********************************************************************)
IF ErrorID = 0 
THEN
	GetAxErrTxt												:= CONCAT(Quelle,'-Kein Fehler vorhanden');
ELSE
	(* Infotext ausgeben *)
	CASE ErrorID OF
	(* TwinCat NC und MC Funktion Fehlergruppen *)
	16#4000..16#4099 :	GetAxErrTxt 						:=CONCAT(  Quelle,',NC Fehler');
                                    						
	16#4100..16#4199 :	GetAxErrTxt 						:=CONCAT(  Quelle,',Kanalfehler');
                                    	
	16#4200..16#42FF :	GetAxErrTxt 						:=CONCAT(  Quelle,',Gruppenfehler');
		CASE ErrorID OF
		16#4220 : GetAxErrTxt 								:= CONCAT( GetAxErrTxt,'-Gruppe nicht fertig / Gruppe nicht bereit für neuen Auftrag');
		16#4221 : GetAxErrTxt 								:= CONCAT( GetAxErrTxt,'-Geforderte Sollgeschwindigkeit ist unzulässig');
		16#4222 : GetAxErrTxt 								:= CONCAT( GetAxErrTxt,'-Geforderte Zielposition ist unzulässig (Masterachse)');
		16#4223 : GetAxErrTxt 								:= CONCAT( GetAxErrTxt,'-Regler- und/oder Vorschubfreigabe nicht vorhanden (Masterachse)');
		16#4225 : GetAxErrTxt 								:= CONCAT( GetAxErrTxt,'-Antriebshardware nicht betriebsbereit bei Achsstart');
		16#4238 : GetAxErrTxt 								:= CONCAT( GetAxErrTxt,'-Geschwindigkeits-Override (StartOverride) unzulässig');
		16#4242 : GetAxErrTxt 								:= CONCAT( GetAxErrTxt,'-Stop ist schon aktiv');
		16#4260 : GetAxErrTxt 								:= CONCAT( GetAxErrTxt,'-Reglerfreigabe nicht vorhanden');
		16#4263 : GetAxErrTxt 								:= CONCAT( GetAxErrTxt,'-Einzelsatz Betrieb (Single Step Mode) es kann kein anderer Auftrag gestartet werden');
                              								
		16#428D : GetAxErrTxt 								:= CONCAT( GetAxErrTxt,'-Ungültiger Abkoppeltyp/Nachstart-Typ');
		16#428E : GetAxErrTxt 								:= CONCAT( GetAxErrTxt,'-Unerlaubte Ziel-Geschwindigkeit beim Abkoppeln einer Slaveachse');
		16#428F : GetAxErrTxt 								:= CONCAT( GetAxErrTxt,'-Aktivierung neue Dynamikparameter kann nicht durchgeführt werden');
		16#4290 : GetAxErrTxt 								:= CONCAT( GetAxErrTxt,'-Kommando kann nicht durchgeführt werden da sich die Achse bereits in der Bemsphase befindet');
		16#42A0 : GetAxErrTxt 								:= CONCAT( GetAxErrTxt,'-Gruppen-/Achsfolgefehler');
		END_CASE

	16#4300..16#4399 :	GetAxErrTxt 						:=CONCAT(  Quelle,',Achsfehler');
		CASE ErrorID OF
		16#4356 : GetAxErrTxt 								:= CONCAT( GetAxErrTxt,'-Reglerfreigabe für Achse nicht vorhanden');
		16#4357 : GetAxErrTxt 								:= CONCAT( GetAxErrTxt,'-Vorschubfrg für negative Verfahrr. nicht vorhanden');
		16#4358 : GetAxErrTxt 								:= CONCAT( GetAxErrTxt,'-Vorschubfrg für positive Verfahrr. nicht vorhanden');
		16#4359 : GetAxErrTxt 								:= CONCAT( GetAxErrTxt,'-Die geforderte Sollgeschw. für einen Pos.auftrag ist nicht erlaubt');
		16#435A : GetAxErrTxt 								:= CONCAT( GetAxErrTxt,'-Verfahrweg kleiner ein Geberinkrement (INTERNER FEHLER) (s. Skalierungsfaktor)');
		16#435B : GetAxErrTxt 								:= CONCAT( GetAxErrTxt,'-Überwachung Sollbeschleunigung (INTERNER FEHLER)');
		16#435C : GetAxErrTxt 								:= CONCAT( GetAxErrTxt,'-PEH-Zeitüberwachung, Zielpos.­fenster nach Pos. nicht erreicht');
		16#435D : GetAxErrTxt 								:= CONCAT( GetAxErrTxt,'-Encoder-Existenz-Überwachung / Bewegungsüberwachung');
		16#435E : GetAxErrTxt 								:= CONCAT( GetAxErrTxt,'-Schleifenweg kleiner als Bremsweg');
		16#43A0 : GetAxErrTxt 								:= CONCAT( GetAxErrTxt,'-Achsfolgefehler');
		END_CASE

	16#4400..16#4499 :	GetAxErrTxt 						:=CONCAT( Quelle, ',Geberfehler');
		CASE ErrorID OF
		16#4460 : GetAxErrTxt 								:= CONCAT( GetAxErrTxt,'-Software Endlage Minimum (Achsstart)');
		16#4461 : GetAxErrTxt 								:= CONCAT( GetAxErrTxt,'-Software Endlage Maximum (Achsstart)');
		16#4462 : GetAxErrTxt 								:= CONCAT( GetAxErrTxt,'-Software Endlage Minimum (Positioniervorgang)');
		16#4463 : GetAxErrTxt 								:= CONCAT( GetAxErrTxt,'-Software Endlage Maximum (Positioniervorgang)');
		END_CASE

	16#4500..16#4599 :	GetAxErrTxt 						:=CONCAT(  Quelle,',Reglerfehler');
		CASE ErrorID OF
		16#4650 : GetAxErrTxt 								:= CONCAT( GetAxErrTxt,'-Antriebshardware nicht betriebsbereit');
		END_CASE

	16#4600..16#4699 :	GetAxErrTxt 						:=CONCAT(  Quelle,',Antriebsfehler');
                                    						
	16#4A00..16#4A99 :	GetAxErrTxt 						:=CONCAT(  Quelle,',Tabellenfehler');
                                    	                	
	16#4B00..16#4B99 :	GetAxErrTxt 						:=CONCAT( Quelle,',NC SPS Fehler');
		CASE ErrorID OF
		16#4B00 : GetAxErrTxt 								:= CONCAT( GetAxErrTxt,'-Achse ist gestoppt worden');
		16#4B01 : GetAxErrTxt 								:= CONCAT( GetAxErrTxt,'-Achse kann nicht gestartet werden');
		16#4B02 : GetAxErrTxt 								:= CONCAT( GetAxErrTxt,'-Kontrollmodus nicht zulässig');
		16#4B03 : GetAxErrTxt 								:= CONCAT( GetAxErrTxt,'-Achse bewegt sich nicht');
		16#4B04 : GetAxErrTxt 								:= CONCAT( GetAxErrTxt,'-Falscher Modus für RestartPosAndVelo');
		16#4B05 : GetAxErrTxt 								:= CONCAT( GetAxErrTxt,'-Befehl nicht zulässig');
		16#4B06 : GetAxErrTxt 								:= CONCAT( GetAxErrTxt,'-Parameter nicht korrekt');
		16#4B07 : GetAxErrTxt 								:= CONCAT( GetAxErrTxt,'-Zielposition Timeout');
		16#4B08 : GetAxErrTxt 								:= CONCAT( GetAxErrTxt,'-Achse ist im geschützten Modus');
		16#4B09 : GetAxErrTxt 								:= CONCAT( GetAxErrTxt,'-Achse ist nicht bereit');
		16#4B0A : GetAxErrTxt 								:= CONCAT( GetAxErrTxt,'-Fehler beim Referenzieren');
		16#4B0B : GetAxErrTxt 								:= CONCAT( GetAxErrTxt,'-Fehlerhafte Definition des Triggereingangs');
		16#4B0C : GetAxErrTxt 								:= CONCAT( GetAxErrTxt,'-Positionslatch wurde deaktiviert');
		(*-----------------------------------*)
		(* 	4B10 .. 4B2F used in NCI context *)
		(*-----------------------------------*)
		(* 	4B30 .. 4B3F used in TcMcCam     *)
		(*  type MC_NC_TableErrorCodes		 *)
		(*-----------------------------------*)
		END_CASE

	ELSE (* case else *)
		GetAxErrTxt 										:= CONCAT(Quelle,',Unbekannte Ax-Fehlergruppe, ID:');
		GetAxErrTxt 										:= CONCAT(GetAxErrTxt,DINT_TO_STRING(ErrorID));
	END_CASE
END_IF

(**********************************************************************************************************)

END_FUNCTION

// ---- POUs/PTP/03_Utilities/MMS_TO_MMIN.TcPOU
FUNCTION MMS_TO_MMIN : LREAL
VAR_INPUT
	IN														:	LREAL;
END_VAR
VAR
END_VAR

MMS_TO_MMIN 												:= IN * 0.001 * 60;

END_FUNCTION

// ---- POUs/UNIT/fb_Apron/FB_FoldAbsPos.TcPOU
FUNCTION_BLOCK FB_FoldAbsPos
VAR_INPUT
	Top_Enable	:BOOL;	
	Top_Target	:REAL;
	Btm_Enable	:BOOL;
	Btm_Target	:REAL;
	AutoFold	:BOOL;	(*true: Auto Fold and Back*)
	Rst	:BOOL;
END_VAR
VAR_OUTPUT
	TopDone	:BOOL;
	BtmDone	:BOOL;
	bOutApronTop_FoldFWD	:BOOL;
	bOutApronTop_FoldBWD	:BOOL;
	bOutApronBtm_FoldFWD	:BOOL;
	bOutApronBtm_FoldBWD	:BOOL;
	bApronFold_AtSlow: INPUT;
END_VAR
VAR
	tMan10,tMan20	:TON;
	iApronBtmFoldAbs: INT;
	iApronTopFoldAbs: INT;

	i2: INT;
	j2: INT;
	i1: INT;
	j1: INT;
	tonTop1: Ton;
	tonBtm1: Ton;
	Btm_Target1,Top_Target1: REAL;
	Btm_Target_Max: REAL;
	Top_Target_Max: REAL;
	
	BB: BOOL;
	tMan11: Ton;
	tMan21: Ton;
	cont: INT := 0;
	minclampress: REAL;
END_VAR

IF Rst THEN
	iApronTopFoldAbs	:=50;
	iApronBtmFoldAbs	:=50;
END_IF

Top_Target_Max:= SEL( stFolder.Status.Clamp_AtZeroPoint,115,147);
Top_Target1:=LIMIT(0, 180-Top_Target,Top_Target_Max);
(*上折弯定位+自由折弯*)
CASE iApronTopFoldAbs OF
	0:
		TopDone	:=FALSE;
		IF Top_Enable THEN
			tMan20(IN:=FALSE);
			IF stFolder.Status.ApronTopSlide_AtWork AND (NOT stFolder.Status.ApronBtmSlide_AtWork) AND stFolder.Status.Slitter_AtHome THEN
				IF Hmi_bArray[43] THEN
					iApronTopFoldAbs:=31;
				ELSIF Top_Target1>stFolder.ApronTop_Fold_ActAngle THEN
					iApronTopFoldAbs:=10;
				ELSIF Top_Target1<stFolder.ApronTop_Fold_ActAngle THEN
					iApronTopFoldAbs:=20;
				ELSE
					iApronTopFoldAbs:=50;
				END_IF
			ELSE
				Hmi_iArray[25]:=Hmi_iArray[25] OR 16#0002;
				iApronTopFoldAbs	:=60;
			END_IF
		END_IF
	10:
		IF stFolder.ApronTop_Fold_ActAngle < Top_Target1 THEN
			bOutApronTop_FoldFWD	:=TRUE;
			bOutApronTop_FoldBWD	:=FALSE;
		ELSE
			IF AutoFold THEN
				iApronTopFoldAbs	:= 30;
			ELSE
				iApronTopFoldAbs	:= 50;
			END_IF
		END_IF;
	20:
		IF stFolder.ApronTop_Fold_ActAngle > Top_Target1 THEN
			bOutApronTop_FoldFWD	:=FALSE;
			bOutApronTop_FoldBWD	:=TRUE;
		END_IF;
		IF stFolder.ApronTop_Fold_ActAngle <= Top_Target1 OR stFolder.Status.ApronTopFold_AtHome THEN
			
			IF AutoFold THEN
				iApronTopFoldAbs	:= 30;
			ELSE
				iApronTopFoldAbs	:= 50;
			END_IF
		END_IF;
	30:
		bOutApronTop_FoldFWD	:=bOutApronTop_FoldBWD	:=FALSE;
		tMan20(IN:=TRUE , PT:=T#200MS , Q=> , ET=> );
		IF NOT stFolder.Status.Flip_WorkDone THEN
			iApronTopFoldAbs	:=SEL(tMan20.Q,30,31);
		END_IF
		
	31:
		IF stFolder.ApronTop_Fold_ActAngle > 0 THEN
			Top_Target1:=0;
			bOutApronTop_FoldFWD	:=FALSE;
			bOutApronTop_FoldBWD	:=TRUE;
		ELSE
			iApronTopFoldAbs	:= 50;
		END_IF
	50:
		bOutApronTop_FoldFWD	:=bOutApronTop_FoldBWD	:=FALSE;
		tMan21(IN:=TRUE , PT:=T#40MS , Q=> , ET=> );	//此处的40ms延迟，不然会有顿响
		IF tMan21.Q THEN
			iApronTopFoldAbs	:= 51;
		END_IF
	51: 
		TopDone	:=TRUE;
		iApronTopFoldAbs	:= 60;
	60:
		iApronTopFoldAbs	:= 0;
		tMan20(IN:=FALSE);tMan21(IN:=FALSE);
		Top_Enable	:=FALSE;
END_CASE




Btm_Target_Max:= SEL( stFolder.Status.Clamp_AtPressPoint,95,147);	//Limit Fold Angle ,when Clamp isn't at PressPoint
Btm_Target1:= LIMIT(0, 180-Btm_Target,Btm_Target_Max);
CASE iApronBtmFoldAbs OF
	0:
		BtmDone	:=FALSE;
		IF Btm_Enable THEN
			tMan10(IN:=false);
			IF stFolder.Status.ApronBtmSlide_AtWork AND (NOT stFolder.Status.ApronTopSlide_AtWork) AND stFolder.Status.Slitter_AtHome THEN
				IF Hmi_bArray[43] THEN	//翻板向下
					iApronBtmFoldAbs:=31;
				ELSIF Btm_Target1>stFolder.ApronBtm_Fold_ActAngle THEN
					iApronBtmFoldAbs:=10;
				ELSIF Btm_Target1<stFolder.ApronBtm_Fold_ActAngle THEN
					iApronBtmFoldAbs:=20;
				ELSE
					iApronBtmFoldAbs:=50;
				END_IF
			ELSE
				Hmi_iArray[25]:=Hmi_iArray[25] OR 16#0008;
				iApronBtmFoldAbs	:=60;
			END_IF
		END_IF
	10:
		IF stFolder.ApronBtm_Fold_ActAngle < Btm_Target1 THEN
			bOutApronBtm_FoldFWD	:=TRUE;
			bOutApronBtm_FoldBWD	:=FALSE;
		ELSE
			IF AutoFold THEN
				iApronBtmFoldAbs	:= 30;
			ELSE
				iApronBtmFoldAbs	:= 50;
			END_IF
		END_IF;
	20:
		IF stFolder.ApronBtm_Fold_ActAngle > Btm_Target1 THEN
			bOutApronBtm_FoldFWD	:=FALSE;
			bOutApronBtm_FoldBWD	:=TRUE;
		END_IF;
		IF stFolder.ApronBtm_Fold_ActAngle <= Btm_Target1 OR stFolder.Status.ApronBtmFold_AtHome THEN
			IF AutoFold THEN
				iApronBtmFoldAbs	:= 30;
			ELSE
				iApronBtmFoldAbs	:= 50;
			END_IF
		END_IF;
	30:
		bOutApronBtm_FoldFWD	:=bOutApronBtm_FoldBWD	:=FALSE;
		tMan10(IN:=TRUE , PT:=T#200MS , Q=> , ET=> );
		iApronBtmFoldAbs	:=SEL(tMan10.Q,30,31);
	31:
		IF stFolder.ApronBtm_Fold_ActAngle <= 0   THEN
			iApronBtmFoldAbs	:= 50;
		ELSE
			Btm_Target1:=0;
			bOutApronBtm_FoldFWD	:=FALSE;
			bOutApronBtm_FoldBWD	:=TRUE;
		END_IF
	50:
		bOutApronBtm_FoldFWD	:=bOutApronBtm_FoldBWD	:=FALSE;
		tMan11(IN:=TRUE , PT:=T#40MS , Q=> , ET=> );				//此处的40ms延迟，不然会有顿响
		IF tMan11.Q THEN
			iApronBtmFoldAbs	:= 51;
		END_IF
	51:		
		BtmDone	:=TRUE;
		iApronBtmFoldAbs	:= 60;
	60:		
		iApronBtmFoldAbs	:= 0;
		tMan10(IN:=FALSE);tMan11(IN:=FALSE);
		Btm_Enable	:=FALSE;
END_CASE

//bApronFold_AtSlow(PT_OFF:=T#50MS);
//IF     (iApronTopFoldAbs>0 AND bOutApronTop_FoldFWD AND stFolder.ApronTop_Fold_ActAngle>110.0 AND ABS(stFolder.ApronTop_Fold_ActAngle-Top_Target1)<CONST_APRON_FOLD_DECWINDOW+20 )
//	OR (iApronTopFoldAbs>0 AND bOutApronTop_FoldFWD AND stFolder.ApronTop_Fold_ActAngle<=110.0 AND ABS(stFolder.ApronTop_Fold_ActAngle-Top_Target1)<CONST_APRON_FOLD_DECWINDOW )
//	OR (iApronTopFoldAbs>0 AND bOutApronTop_FoldBWD AND ABS(stFolder.ApronTop_Fold_ActAngle-Top_Target1)<CONST_APRON_FOLD_DECWINDOW+29 )
//	OR (iApronBtmFoldAbs>0 AND bOutApronBtm_FoldFWD AND stFolder.ApronBtm_Fold_ActAngle>110.0 AND ABS(stFolder.ApronBtm_Fold_ActAngle-Btm_Target1)<CONST_APRON_FOLD_DECWINDOW+20) 
//	OR (iApronBtmFoldAbs>0 AND bOutApronBtm_FoldFWD AND stFolder.ApronBtm_Fold_ActAngle<=110.0 AND  ABS(stFolder.ApronBtm_Fold_ActAngle-Btm_Target1)<CONST_APRON_FOLD_DECWINDOW)
//	OR (iApronBtmFoldAbs>0 AND bOutApronBtm_FoldBWD AND ABS(stFolder.ApronBtm_Fold_ActAngle-Btm_Target1)<CONST_APRON_FOLD_DECWINDOW+28) 
//THEN
//	bApronFold_AtSlow.INPUT	:=TRUE;
			
//ELSE
//	bApronFold_AtSlow.INPUT	:=FALSE;
//END_IF

bApronFold_AtSlow(PT_OFF:=T#50MS);
IF (iApronTopFoldAbs>0 AND bOutApronTop_FoldFWD AND stFolder.ApronTop_Fold_ActAngle>110.0 AND ABS(stFolder.ApronTop_Fold_ActAngle-Top_Target1)< CNST_APRON_TOPFOLD_BWD_DecDis )
	OR (iApronTopFoldAbs>0 AND bOutApronTop_FoldFWD AND stFolder.ApronTop_Fold_ActAngle<=110.0 AND ABS(stFolder.ApronTop_Fold_ActAngle-Top_Target1)<CNST_APRON_TOPFOLD_FWD_DecDis_LE110 )
	OR (iApronTopFoldAbs>0 AND bOutApronTop_FoldBWD AND ABS(stFolder.ApronTop_Fold_ActAngle-Top_Target1)<CNST_APRON_TOPFOLD_BWD_DecDis )
	OR (iApronBtmFoldAbs>0 AND bOutApronBtm_FoldFWD AND stFolder.ApronBtm_Fold_ActAngle>110.0 AND ABS(stFolder.ApronBtm_Fold_ActAngle-Btm_Target1)<CNST_APRON_BTMFOLD_FWD_DecDis_GT110) 
	OR (iApronBtmFoldAbs>0 AND bOutApronBtm_FoldFWD AND stFolder.ApronBtm_Fold_ActAngle<=110.0 AND  ABS(stFolder.ApronBtm_Fold_ActAngle-Btm_Target1)<CNST_APRON_BTMFOLD_FWD_DecDis_LE110)
	OR (iApronBtmFoldAbs>0 AND bOutApronBtm_FoldBWD AND ABS(stFolder.ApronBtm_Fold_ActAngle-Btm_Target1)<CNST_APRON_BTMFOLD_BWD_DecDis ) 
THEN
	bApronFold_AtSlow.INPUT	:=TRUE;
ELSE
	bApronFold_AtSlow.INPUT	:=FALSE;
END_IF
	





tonTop1(IN:=TopDone , PT:=T#500MS , Q=> , ET=> );
IF tonTop1.Q THEN
	TopDone	:=FALSE;
END_IF;
tonBtm1(IN:=BtmDone , PT:=T#500MS , Q=> , ET=> );
IF tonBtm1.Q THEN
	BtmDone	:=FALSE;
END_IF

END_FUNCTION_BLOCK

